    - target stk_p2_s18_t7 (Cartesian target) at (974.5, -259.38, 673.26) mm, rotated rx -64.06 ry 82.47 rz -57.48 deg; joints [17.675, -65.878, 133.528, 25.602, -72.986, -2.699] of KR 8 1620 ARC HW
    - target stk_p2_s18_t8 (Cartesian target) at (974.72, -248.82, 673.38) mm, rotated rx -62.73 ry 82.82 rz -56.53 deg; joints [16.995, -66.047, 133.813, 24.489, -72.919, -2.65] of KR 8 1620 ARC HW
    - target stk_p2_s18_t9 (Cartesian target) at (974.93, -238.26, 673.5) mm, rotated rx -61.27 ry 83.16 rz -55.44 deg; joints [16.309, -66.209, 134.087, 23.369, -72.854, -2.602] of KR 8 1620 ARC HW
    - target stk_p2_s18_t10 (Cartesian target) at (975.15, -227.7, 673.63) mm, rotated rx -59.65 ry 83.5 rz -54.2 deg; joints [15.619, -66.365, 134.348, 22.243, -72.793, -2.556] of KR 8 1620 ARC HW
    - target stk_p2_s18_t11 (Cartesian target) at (975.37, -217.15, 673.75) mm, rotated rx -57.85 ry 83.83 rz -52.78 deg; joints [14.924, -66.514, 134.596, 21.111, -72.734, -2.512] of KR 8 1620 ARC HW
    - target stk_p2_s18_t12 (Cartesian target) at (975.59, -206.59, 673.87) mm, rotated rx -55.85 ry 84.16 rz -51.15 deg; joints [14.225, -66.656, 134.833, 19.974, -72.677, -2.468] of KR 8 1620 ARC HW
    - target stk_p2_s18_t13 (Cartesian target) at (975.81, -196.03, 674) mm, rotated rx -53.61 ry 84.48 rz -49.29 deg; joints [13.522, -66.791, 135.056, 18.832, -72.624, -2.426] of KR 8 1620 ARC HW
    - target stk_p2_s18_t14 (Cartesian target) at (976.03, -185.47, 674.12) mm, rotated rx -51.1 ry 84.79 rz -47.16 deg; joints [12.814, -66.92, 135.267, 17.684, -72.573, -2.385] of KR 8 1620 ARC HW
    - target stk_p2_s18_t15 (Cartesian target) at (976.25, -174.91, 674.24) mm, rotated rx -48.28 ry 85.09 rz -44.71 deg; joints [12.103, -67.041, 135.466, 16.531, -72.525, -2.344] of KR 8 1620 ARC HW
    - target stk_p2_s18_t16 (Cartesian target) at (976.47, -164.35, 674.37) mm, rotated rx -45.1 ry 85.37 rz -41.91 deg; joints [11.388, -67.155, 135.652, 15.374, -72.479, -2.305] of KR 8 1620 ARC HW
    - target stk_p2_s18_t17 (Cartesian target) at (976.69, -153.8, 674.49) mm, rotated rx -41.5 ry 85.64 rz -38.69 deg; joints [10.669, -67.262, 135.825, 14.213, -72.437, -2.266] of KR 8 1620 ARC HW
    - target stk_p2_s18_t18 (Cartesian target) at (976.91, -143.24, 674.61) mm, rotated rx -37.45 ry 85.89 rz -35.02 deg; joints [9.947, -67.362, 135.985, 13.048, -72.397, -2.228] of KR 8 1620 ARC HW
    - target stk_p2_s18_t19 (Cartesian target) at (977.13, -132.68, 674.74) mm, rotated rx -32.89 ry 86.12 rz -30.84 deg; joints [9.223, -67.455, 136.132, 11.878, -72.359, -2.191] of KR 8 1620 ARC HW
    - target stk_p2_s18_t20 (Cartesian target) at (977.35, -122.12, 674.86) mm, rotated rx -27.79 ry 86.32 rz -26.12 deg; joints [8.495, -67.54, 136.267, 10.706, -72.324, -2.154] of KR 8 1620 ARC HW
    - target stk_p2_s18_t21 (Cartesian target) at (977.57, -111.56, 674.99) mm, rotated rx -22.15 ry 86.49 rz -20.87 deg; joints [7.765, -67.618, 136.388, 9.53, -72.292, -2.118] of KR 8 1620 ARC HW
    - target stk_p2_s18_t22 (Cartesian target) at (977.79, -101, 675.11) mm, rotated rx -16.01 ry 86.62 rz -15.1 deg; joints [7.032, -67.689, 136.497, 8.351, -72.263, -2.082] of KR 8 1620 ARC HW
    - target stk_p2_s18_t23 (Cartesian target) at (978.01, -90.44, 675.23) mm, rotated rx -9.44 ry 86.71 rz -8.92 deg; joints [6.298, -67.752, 136.592, 7.17, -72.236, -2.047] of KR 8 1620 ARC HW
    - target stk_p2_s18_t24 (Cartesian target) at (978.22, -79.89, 675.36) mm, rotated rx -2.6 ry 86.76 rz -2.46 deg; joints [5.561, -67.807, 136.675, 5.986, -72.212, -2.011] of KR 8 1620 ARC HW
    - target stk_p2_s18_t25 (Cartesian target) at (978.44, -69.33, 675.48) mm, rotated rx 4.34 ry 86.76 rz 4.1 deg; joints [4.823, -67.856, 136.745, 4.801, -72.191, -1.976] of KR 8 1620 ARC HW
    - target stk_p2_s19_t0 (Cartesian target) at (980.09, -20.25, 992.92) mm, rotated rx 166.42 ry 81.24 rz 164.19 deg; joints [1.382, -82.788, 120.669, -1.392, -29.376, -0.961] of KR 8 1620 ARC HW
    - target stk_p2_s19_t0 (Cartesian target) at (980.09, -20.25, 992.92) mm, rotated rx 166.42 ry 81.24 rz 164.19 deg; joints [1.382, -82.788, 120.669, -1.392, -29.376, -0.961] of KR 8 1620 ARC HW
    - target stk_p2_s19_t1 (Cartesian target) at (980.31, -9.7, 993.04) mm, rotated rx 163.97 ry 81.14 rz 161.32 deg; joints [0.646, -82.79, 120.662, -3.667, -29.403, 0.461] of KR 8 1620 ARC HW
    - target stk_p2_s19_t2 (Cartesian target) at (980.53, 0.86, 993.17) mm, rotated rx 161.59 ry 81.02 rz 158.52 deg; joints [-0.09, -82.781, 120.643, -5.935, -29.465, 1.877] of KR 8 1620 ARC HW
    - target stk_p2_s19_t3 (Cartesian target) at (980.75, 11.42, 993.29) mm, rotated rx 159.27 ry 80.89 rz 155.78 deg; joints [-0.826, -82.763, 120.613, -8.193, -29.56, 3.283] of KR 8 1620 ARC HW
    - target stk_p2_s19_t4 (Cartesian target) at (980.97, 21.98, 993.41) mm, rotated rx 157.02 ry 80.74 rz 153.11 deg; joints [-1.561, -82.735, 120.571, -10.434, -29.689, 4.673] of KR 8 1620 ARC HW
    - target stk_p2_s19_t5 (Cartesian target) at (981.19, 32.54, 993.54) mm, rotated rx 154.85 ry 80.58 rz 150.52 deg; joints [-2.295, -82.696, 120.518, -12.654, -29.85, 6.042] of KR 8 1620 ARC HW
    - target stk_p2_s19_t6 (Cartesian target) at (981.41, 43.1, 993.66) mm, rotated rx 152.76 ry 80.4 rz 148 deg; joints [-3.028, -82.648, 120.453, -14.85, -30.044, 7.388] of KR 8 1620 ARC HW
    - target stk_p2_s19_t7 (Cartesian target) at (981.63, 53.65, 993.78) mm, rotated rx 150.74 ry 80.21 rz 145.56 deg; joints [-3.76, -82.589, 120.376, -17.016, -30.269, 8.706] of KR 8 1620 ARC HW
    - target stk_p2_s19_t8 (Cartesian target) at (981.85, 64.21, 993.91) mm, rotated rx 148.8 ry 80.02 rz 143.2 deg; joints [-4.489, -82.521, 120.288, -19.15, -30.525, 9.992] of KR 8 1620 ARC HW
    - target stk_p2_s19_t9 (Cartesian target) at (982.07, 74.77, 994.03) mm, rotated rx 146.94 ry 79.81 rz 140.92 deg; joints [-5.218, -82.442, 120.188, -21.248, -30.81, 11.243] of KR 8 1620 ARC HW
    - target stk_p2_s19_t10 (Cartesian target) at (982.29, 85.33, 994.15) mm, rotated rx 145.16 ry 79.59 rz 138.72 deg; joints [-5.943, -82.354, 120.077, -23.307, -31.124, 12.457] of KR 8 1620 ARC HW
    - target stk_p2_s19_t11 (Cartesian target) at (982.5, 95.89, 994.28) mm, rotated rx 143.45 ry 79.36 rz 136.59 deg; joints [-6.667, -82.256, 119.954, -25.325, -31.465, 13.632] of KR 8 1620 ARC HW
    - target stk_p2_s19_t12 (Cartesian target) at (982.72, 106.45, 994.4) mm, rotated rx 141.82 ry 79.13 rz 134.54 deg; joints [-7.388, -82.148, 119.82, -27.301, -31.831, 14.766] of KR 8 1620 ARC HW
    - target stk_p2_s19_t13 (Cartesian target) at (982.94, 117.01, 994.52) mm, rotated rx 140.26 ry 78.88 rz 132.56 deg; joints [-8.106, -82.031, 119.674, -29.232, -32.222, 15.858] of KR 8 1620 ARC HW
    - target stk_p2_s19_t14 (Cartesian target) at (983.16, 127.56, 994.65) mm, rotated rx 138.76 ry 78.63 rz 130.65 deg; joints [-8.821, -81.904, 119.517, -31.118, -32.637, 16.906] of KR 8 1620 ARC HW
    - target stk_p2_s19_t15 (Cartesian target) at (983.38, 138.12, 994.77) mm, rotated rx 137.34 ry 78.38 rz 128.81 deg; joints [-9.533, -81.768, 119.348, -32.958, -33.073, 17.91] of KR 8 1620 ARC HW
    - target stk_p2_s19_t16 (Cartesian target) at (983.6, 148.68, 994.89) mm, rotated rx 135.98 ry 78.11 rz 127.03 deg; joints [-10.241, -81.622, 119.167, -34.751, -33.531, 18.869] of KR 8 1620 ARC HW
    - target stk_p2_s19_t17 (Cartesian target) at (983.82, 159.24, 995.02) mm, rotated rx 134.68 ry 77.84 rz 125.32 deg; joints [-10.946, -81.466, 118.975, -36.498, -34.008, 19.785] of KR 8 1620 ARC HW
    - target stk_p2_s19_t18 (Cartesian target) at (984.04, 169.8, 995.14) mm, rotated rx 133.43 ry 77.57 rz 123.66 deg; joints [-11.647, -81.302, 118.772, -38.198, -34.503, 20.657] of KR 8 1620 ARC HW
    - target stk_p2_s19_t19 (Cartesian target) at (984.26, 180.36, 995.27) mm, rotated rx 132.25 ry 77.29 rz 122.06 deg; joints [-12.344, -81.128, 118.557, -39.852, -35.015, 21.485] of KR 8 1620 ARC HW
    - target stk_p2_s19_t20 (Cartesian target) at (984.48, 190.91, 995.39) mm, rotated rx 131.11 ry 77 rz 120.51 deg; joints [-13.036, -80.945, 118.33, -41.461, -35.542, 22.271] of KR 8 1620 ARC HW
    - target stk_p2_s19_t21 (Cartesian target) at (984.7, 201.47, 995.51) mm, rotated rx 130.03 ry 76.71 rz 119.02 deg; joints [-13.725, -80.753, 118.092, -43.024, -36.084, 23.015] of KR 8 1620 ARC HW
    - target stk_p2_s19_t22 (Cartesian target) at (984.92, 212.03, 995.64) mm, rotated rx 128.99 ry 76.42 rz 117.57 deg; joints [-14.408, -80.553, 117.842, -44.544, -36.64, 23.718] of KR 8 1620 ARC HW
    - target stk_p2_s19_t23 (Cartesian target) at (985.14, 222.59, 995.76) mm, rotated rx 128 ry 76.12 rz 116.17 deg; joints [-15.087, -80.343, 117.581, -46.021, -37.208, 24.382] of KR 8 1620 ARC HW
    - target stk_p2_s19_t24 (Cartesian target) at (985.36, 233.15, 995.88) mm, rotated rx 127.06 ry 75.83 rz 114.81 deg; joints [-15.761, -80.125, 117.309, -47.456, -37.787, 25.008] of KR 8 1620 ARC HW
    - target stk_p2_s19_t25 (Cartesian target) at (985.58, 243.71, 996.01) mm, rotated rx 126.15 ry 75.52 rz 113.5 deg; joints [-16.43, -79.898, 117.025, -48.85, -38.376, 25.597] of KR 8 1620 ARC HW
    - target stk_p2_s20_t0 (Cartesian target) at (973.51, -337.01, 989.21) mm, rotated rx -130.97 ry 77.39 rz -120.69 deg; joints [22.363, -78.272, 115.517, 53.029, -40.963, -30.398] of KR 8 1620 ARC HW
    - target stk_p2_s20_t0 (Cartesian target) at (973.51, -337.01, 989.21) mm, rotated rx -130.97 ry 77.39 rz -120.69 deg; joints [22.363, -78.272, 115.517, 53.029, -40.963, -30.398] of KR 8 1620 ARC HW
    - target stk_p2_s20_t1 (Cartesian target) at (973.73, -326.45, 989.34) mm, rotated rx -132.16 ry 77.66 rz -122.29 deg; joints [21.726, -78.55, 115.855, 51.798, -40.347, -29.959] of KR 8 1620 ARC HW
    - target stk_p2_s20_t2 (Cartesian target) at (973.95, -315.89, 989.46) mm, rotated rx -133.41 ry 77.93 rz -123.94 deg; joints [21.084, -78.821, 116.182, 50.533, -39.738, -29.489] of KR 8 1620 ARC HW
    - target stk_p2_s20_t3 (Cartesian target) at (974.17, -305.33, 989.58) mm, rotated rx -134.71 ry 78.2 rz -125.65 deg; joints [20.436, -79.083, 116.497, 49.231, -39.135, -28.988] of KR 8 1620 ARC HW
    - target stk_p2_s20_t4 (Cartesian target) at (974.39, -294.77, 989.71) mm, rotated rx -136.07 ry 78.46 rz -127.42 deg; joints [19.783, -79.337, 116.8, 47.892, -38.541, -28.453] of KR 8 1620 ARC HW
    - target stk_p2_s20_t5 (Cartesian target) at (974.61, -284.21, 989.83) mm, rotated rx -137.5 ry 78.71 rz -129.26 deg; joints [19.124, -79.583, 117.093, 46.515, -37.955, -27.884] of KR 8 1620 ARC HW
    - target stk_p2_s20_t6 (Cartesian target) at (974.83, -273.66, 989.95) mm, rotated rx -139 ry 78.95 rz -131.17 deg; joints [18.46, -79.821, 117.374, 45.098, -37.378, -27.279] of KR 8 1620 ARC HW
    - target stk_p2_s20_t7 (Cartesian target) at (975.05, -263.1, 990.08) mm, rotated rx -140.57 ry 79.19 rz -133.15 deg; joints [17.791, -80.05, 117.643, 43.64, -36.812, -26.637] of KR 8 1620 ARC HW
    - target stk_p2_s20_t8 (Cartesian target) at (975.27, -252.54, 990.2) mm, rotated rx -142.2 ry 79.43 rz -135.2 deg; joints [17.116, -80.271, 117.901, 42.14, -36.258, -25.955] of KR 8 1620 ARC HW
    - target stk_p2_s20_t9 (Cartesian target) at (975.49, -241.98, 990.32) mm, rotated rx -143.91 ry 79.65 rz -137.32 deg; joints [16.437, -80.484, 118.148, 40.597, -35.716, -25.234] of KR 8 1620 ARC HW
    - target stk_p2_s20_t10 (Cartesian target) at (975.71, -231.42, 990.45) mm, rotated rx -145.7 ry 79.86 rz -139.53 deg; joints [15.754, -80.687, 118.383, 39.01, -35.188, -24.472] of KR 8 1620 ARC HW
    - target stk_p2_s20_t11 (Cartesian target) at (975.93, -220.86, 990.57) mm, rotated rx -147.57 ry 80.07 rz -141.81 deg; joints [15.065, -80.882, 118.606, 37.378, -34.675, -23.668] of KR 8 1620 ARC HW
    - target stk_p2_s20_t12 (Cartesian target) at (976.14, -210.31, 990.69) mm, rotated rx -149.51 ry 80.26 rz -144.16 deg; joints [14.373, -81.068, 118.819, 35.7, -34.178, -22.821] of KR 8 1620 ARC HW
    - target stk_p2_s20_t13 (Cartesian target) at (976.36, -199.75, 990.82) mm, rotated rx -151.53 ry 80.44 rz -146.6 deg; joints [13.676, -81.244, 119.019, 33.976, -33.698, -21.93] of KR 8 1620 ARC HW
    - target stk_p2_s20_t14 (Cartesian target) at (976.58, -189.19, 990.94) mm, rotated rx -153.63 ry 80.61 rz -149.12 deg; joints [12.975, -81.412, 119.209, 32.206, -33.237, -20.996] of KR 8 1620 ARC HW
    - target stk_p2_s20_t15 (Cartesian target) at (976.8, -178.63, 991.06) mm, rotated rx -155.8 ry 80.77 rz -151.71 deg; joints [12.27, -81.57, 119.386, 30.39, -32.795, -20.017] of KR 8 1620 ARC HW
    - target stk_p2_s20_t16 (Cartesian target) at (977.02, -168.07, 991.19) mm, rotated rx -158.06 ry 80.91 rz -154.38 deg; joints [11.561, -81.719, 119.553, 28.527, -32.375, -18.994] of KR 8 1620 ARC HW
    - target stk_p2_s20_t17 (Cartesian target) at (977.24, -157.51, 991.31) mm, rotated rx -160.38 ry 81.04 rz -157.12 deg; joints [10.849, -81.859, 119.707, 26.619, -31.977, -17.927] of KR 8 1620 ARC HW
    - target stk_p2_s20_t18 (Cartesian target) at (977.46, -146.96, 991.44) mm, rotated rx -162.76 ry 81.16 rz -159.93 deg; joints [10.134, -81.989, 119.851, 24.665, -31.603, -16.817] of KR 8 1620 ARC HW
    - target stk_p2_s20_t19 (Cartesian target) at (977.68, -136.4, 991.56) mm, rotated rx -165.21 ry 81.26 rz -162.8 deg; joints [9.416, -82.11, 119.982, 22.669, -31.254, -15.666] of KR 8 1620 ARC HW
    - target stk_p2_s20_t20 (Cartesian target) at (977.9, -125.84, 991.68) mm, rotated rx -167.71 ry 81.34 rz -165.72 deg; joints [8.695, -82.221, 120.103, 20.631, -30.931, -14.474] of KR 8 1620 ARC HW
    - target stk_p2_s20_t21 (Cartesian target) at (978.12, -115.28, 991.81) mm, rotated rx -170.26 ry 81.41 rz -168.69 deg; joints [7.971, -82.322, 120.211, 18.553, -30.635, -13.243] of KR 8 1620 ARC HW
    - target stk_p2_s20_t22 (Cartesian target) at (978.34, -104.72, 991.93) mm, rotated rx -172.85 ry 81.46 rz -171.7 deg; joints [7.245, -82.413, 120.308, 16.437, -30.369, -11.977] of KR 8 1620 ARC HW
    - target stk_p2_s20_t23 (Cartesian target) at (978.56, -94.16, 992.05) mm, rotated rx -175.46 ry 81.5 rz -174.73 deg; joints [6.517, -82.495, 120.394, 14.288, -30.132, -10.677] of KR 8 1620 ARC HW
    - target stk_p2_s20_t24 (Cartesian target) at (978.78, -83.6, 992.18) mm, rotated rx -178.09 ry 81.51 rz -177.78 deg; joints [5.787, -82.567, 120.468, 12.107, -29.925, -9.347] of KR 8 1620 ARC HW
    - target stk_p2_s20_t25 (Cartesian target) at (979, -73.05, 992.3) mm, rotated rx 179.28 ry 81.51 rz 179.17 deg; joints [5.056, -82.629, 120.53, 9.9, -29.751, -7.991] of KR 8 1620 ARC HW
    - target stk_p3_s21_t0 (Cartesian target) at (979.69, -17.53, 760.58) mm, rotated rx 88.12 ry 87.83 rz 85.95 deg; joints [0.159, -73.03, 133.853, -2.305, -60.913, -1.05] of KR 8 1620 ARC HW
    - target stk_p3_s21_t0 (Cartesian target) at (979.69, -17.53, 760.58) mm, rotated rx 88.12 ry 87.83 rz 85.95 deg; joints [0.159, -73.03, 133.853, -2.305, -60.913, -1.05] of KR 8 1620 ARC HW
    - target stk_p3_s21_t1 (Cartesian target) at (979.91, -6.97, 760.71) mm, rotated rx 88.51 ry 87.43 rz 85.95 deg; joints [-0.582, -73.021, 133.814, -3.603, -60.908, -0.808] of KR 8 1620 ARC HW
    - target stk_p3_s21_t2 (Cartesian target) at (980.13, 3.59, 760.83) mm, rotated rx 88.8 ry 87.04 rz 85.84 deg; joints [-1.323, -73.002, 133.762, -4.901, -60.911, -0.567] of KR 8 1620 ARC HW
    - target stk_p3_s21_t3 (Cartesian target) at (980.35, 14.15, 760.95) mm, rotated rx 89.02 ry 86.65 rz 85.67 deg; joints [-2.063, -72.975, 133.697, -6.197, -60.922, -0.324] of KR 8 1620 ARC HW
    - target stk_p3_s21_t4 (Cartesian target) at (980.56, 24.71, 761.08) mm, rotated rx 89.19 ry 86.26 rz 85.45 deg; joints [-2.801, -72.94, 133.619, -7.492, -60.942, -0.082] of KR 8 1620 ARC HW
    - target stk_p3_s21_t5 (Cartesian target) at (980.78, 35.26, 761.2) mm, rotated rx 89.33 ry 85.86 rz 85.2 deg; joints [-3.538, -72.895, 133.529, -8.784, -60.97, 0.16] of KR 8 1620 ARC HW
    - target stk_p3_s21_t6 (Cartesian target) at (981, 45.82, 761.32) mm, rotated rx 89.45 ry 85.47 rz 84.92 deg; joints [-4.273, -72.843, 133.426, -10.073, -61.007, 0.401] of KR 8 1620 ARC HW
    - target stk_p3_s21_t7 (Cartesian target) at (981.22, 56.38, 761.45) mm, rotated rx 89.55 ry 85.08 rz 84.63 deg; joints [-5.006, -72.781, 133.311, -11.359, -61.051, 0.642] of KR 8 1620 ARC HW
    - target stk_p3_s21_t8 (Cartesian target) at (981.44, 66.94, 761.57) mm, rotated rx 89.63 ry 84.69 rz 84.32 deg; joints [-5.736, -72.712, 133.182, -12.64, -61.104, 0.882] of KR 8 1620 ARC HW
    - target stk_p3_s21_t9 (Cartesian target) at (981.66, 77.5, 761.69) mm, rotated rx 89.7 ry 84.3 rz 84 deg; joints [-6.464, -72.634, 133.042, -13.918, -61.165, 1.122] of KR 8 1620 ARC HW
    - target stk_p3_s21_t10 (Cartesian target) at (981.88, 88.06, 761.82) mm, rotated rx 89.76 ry 83.91 rz 83.67 deg; joints [-7.189, -72.547, 132.888, -15.19, -61.235, 1.36] of KR 8 1620 ARC HW
    - target stk_p3_s21_t11 (Cartesian target) at (982.1, 98.62, 761.94) mm, rotated rx 89.82 ry 83.52 rz 83.34 deg; joints [-7.911, -72.452, 132.722, -16.458, -61.312, 1.597] of KR 8 1620 ARC HW
    - target stk_p3_s21_t12 (Cartesian target) at (982.32, 109.17, 762.07) mm, rotated rx 89.87 ry 83.13 rz 83 deg; joints [-8.629, -72.35, 132.544, -17.72, -61.397, 1.832] of KR 8 1620 ARC HW
    - target stk_p3_s21_t13 (Cartesian target) at (982.54, 119.73, 762.19) mm, rotated rx 89.91 ry 82.74 rz 82.65 deg; joints [-9.344, -72.238, 132.353, -18.975, -61.49, 2.066] of KR 8 1620 ARC HW
    - target stk_p3_s21_t14 (Cartesian target) at (982.76, 130.29, 762.31) mm, rotated rx 89.95 ry 82.35 rz 82.3 deg; joints [-10.055, -72.119, 132.15, -20.224, -61.59, 2.298] of KR 8 1620 ARC HW
    - target stk_p3_s21_t15 (Cartesian target) at (982.98, 140.85, 762.44) mm, rotated rx 89.98 ry 81.97 rz 81.95 deg; joints [-10.763, -71.992, 131.935, -21.467, -61.698, 2.528] of KR 8 1620 ARC HW
    - target stk_p3_s21_t16 (Cartesian target) at (983.2, 151.41, 762.56) mm, rotated rx 90.02 ry 81.58 rz 81.59 deg; joints [-11.466, -71.857, 131.707, -22.702, -61.813, 2.756] of KR 8 1620 ARC HW
    - target stk_p3_s21_t17 (Cartesian target) at (983.42, 161.97, 762.68) mm, rotated rx 90.05 ry 81.19 rz 81.24 deg; joints [-12.165, -71.714, 131.467, -23.929, -61.936, 2.982] of KR 8 1620 ARC HW
    - target stk_p3_s21_t18 (Cartesian target) at (983.64, 172.52, 762.81) mm, rotated rx 90.07 ry 80.81 rz 80.88 deg; joints [-12.86, -71.563, 131.215, -25.149, -62.066, 3.206] of KR 8 1620 ARC HW
    - target stk_p3_s21_t19 (Cartesian target) at (983.85, 183.08, 762.93) mm, rotated rx 90.1 ry 80.42 rz 80.52 deg; joints [-13.55, -71.405, 130.951, -26.361, -62.203, 3.428] of KR 8 1620 ARC HW
    - target stk_p3_s21_t20 (Cartesian target) at (984.07, 193.64, 763.05) mm, rotated rx 90.12 ry 80.04 rz 80.15 deg; joints [-14.235, -71.239, 130.675, -27.563, -62.346, 3.647] of KR 8 1620 ARC HW
    - target stk_p3_s21_t21 (Cartesian target) at (984.29, 204.2, 763.18) mm, rotated rx 90.14 ry 79.65 rz 79.79 deg; joints [-14.915, -71.065, 130.387, -28.758, -62.496, 3.864] of KR 8 1620 ARC HW
    - target stk_p3_s21_t22 (Cartesian target) at (984.51, 214.76, 763.3) mm, rotated rx 90.16 ry 79.27 rz 79.43 deg; joints [-15.59, -70.884, 130.087, -29.943, -62.653, 4.079] of KR 8 1620 ARC HW
    - target stk_p3_s21_t23 (Cartesian target) at (984.73, 225.32, 763.42) mm, rotated rx 90.18 ry 78.89 rz 79.06 deg; joints [-16.259, -70.696, 129.775, -31.118, -62.816, 4.291] of KR 8 1620 ARC HW
    - target stk_p3_s21_t24 (Cartesian target) at (984.95, 235.88, 763.55) mm, rotated rx 90.19 ry 78.51 rz 78.7 deg; joints [-16.924, -70.5, 129.451, -32.284, -62.986, 4.5] of KR 8 1620 ARC HW
    - target stk_p3_s21_t25 (Cartesian target) at (985.17, 246.43, 763.67) mm, rotated rx 90.21 ry 78.13 rz 78.33 deg; joints [-17.583, -70.298, 129.116, -33.441, -63.161, 4.708] of KR 8 1620 ARC HW
    - target stk_p3_s22_t0 (Cartesian target) at (973.11, -334.28, 756.88) mm, rotated rx -88.75 ry 80.51 rz -79.28 deg; joints [21.555, -69.45, 129.11, 34.827, -64.553, -7.278] of KR 8 1620 ARC HW
    - target stk_p3_s22_t0 (Cartesian target) at (973.11, -334.28, 756.88) mm, rotated rx -88.75 ry 80.51 rz -79.28 deg; joints [21.555, -69.45, 129.11, 34.827, -64.553, -7.278] of KR 8 1620 ARC HW
    - target stk_p3_s22_t1 (Cartesian target) at (973.33, -323.72, 757) mm, rotated rx -88.73 ry 80.89 rz -79.64 deg; joints [20.901, -69.681, 129.449, 33.7, -64.344, -7.114] of KR 8 1620 ARC HW
    - target stk_p3_s22_t2 (Cartesian target) at (973.55, -313.16, 757.12) mm, rotated rx -88.7 ry 81.27 rz -79.99 deg; joints [20.24, -69.905, 129.775, 32.562, -64.139, -6.946] of KR 8 1620 ARC HW
    - target stk_p3_s22_t3 (Cartesian target) at (973.77, -302.6, 757.25) mm, rotated rx -88.67 ry 81.65 rz -80.34 deg; joints [19.574, -70.122, 130.09, 31.415, -63.939, -6.776] of KR 8 1620 ARC HW
    - target stk_p3_s22_t4 (Cartesian target) at (973.99, -292.05, 757.37) mm, rotated rx -88.64 ry 82.03 rz -80.69 deg; joints [18.903, -70.332, 130.392, 30.258, -63.745, -6.602] of KR 8 1620 ARC HW
    - target stk_p3_s22_t5 (Cartesian target) at (974.2, -281.49, 757.49) mm, rotated rx -88.61 ry 82.42 rz -81.04 deg; joints [18.226, -70.535, 130.682, 29.092, -63.555, -6.426] of KR 8 1620 ARC HW
    - target stk_p3_s22_t6 (Cartesian target) at (974.42, -270.93, 757.62) mm, rotated rx -88.57 ry 82.8 rz -81.38 deg; joints [17.544, -70.73, 130.96, 27.916, -63.37, -6.246] of KR 8 1620 ARC HW
    - target stk_p3_s22_t7 (Cartesian target) at (974.64, -260.37, 757.74) mm, rotated rx -88.52 ry 83.19 rz -81.72 deg; joints [16.858, -70.918, 131.225, 26.731, -63.19, -6.063] of KR 8 1620 ARC HW
    - target stk_p3_s22_t8 (Cartesian target) at (974.86, -249.81, 757.86) mm, rotated rx -88.47 ry 83.57 rz -82.06 deg; joints [16.166, -71.099, 131.478, 25.537, -63.016, -5.877] of KR 8 1620 ARC HW
    - target stk_p3_s22_t9 (Cartesian target) at (975.08, -239.25, 757.99) mm, rotated rx -88.42 ry 83.96 rz -82.39 deg; joints [15.47, -71.272, 131.719, 24.334, -62.848, -5.687] of KR 8 1620 ARC HW
    - target stk_p3_s22_t10 (Cartesian target) at (975.3, -228.7, 758.11) mm, rotated rx -88.36 ry 84.35 rz -82.71 deg; joints [14.77, -71.437, 131.947, 23.124, -62.686, -5.495] of KR 8 1620 ARC HW
    - target stk_p3_s22_t11 (Cartesian target) at (975.52, -218.14, 758.24) mm, rotated rx -88.28 ry 84.73 rz -83.03 deg; joints [14.065, -71.595, 132.163, 21.905, -62.529, -5.299] of KR 8 1620 ARC HW
    - target stk_p3_s22_t12 (Cartesian target) at (975.74, -207.58, 758.36) mm, rotated rx -88.2 ry 85.12 rz -83.33 deg; joints [13.356, -71.745, 132.367, 20.678, -62.379, -5.099] of KR 8 1620 ARC HW
    - target stk_p3_s22_t13 (Cartesian target) at (975.96, -197.02, 758.48) mm, rotated rx -88.1 ry 85.51 rz -83.62 deg; joints [12.643, -71.887, 132.558, 19.444, -62.235, -4.897] of KR 8 1620 ARC HW
    - target stk_p3_s22_t14 (Cartesian target) at (976.18, -186.46, 758.61) mm, rotated rx -87.98 ry 85.9 rz -83.89 deg; joints [11.927, -72.021, 132.736, 18.202, -62.098, -4.691] of KR 8 1620 ARC HW
    - target stk_p3_s22_t15 (Cartesian target) at (976.4, -175.9, 758.73) mm, rotated rx -87.84 ry 86.29 rz -84.14 deg; joints [11.207, -72.147, 132.901, 16.954, -61.968, -4.482] of KR 8 1620 ARC HW
    - target stk_p3_s22_t16 (Cartesian target) at (976.62, -165.35, 758.85) mm, rotated rx -87.67 ry 86.68 rz -84.35 deg; joints [10.484, -72.265, 133.054, 15.7, -61.844, -4.27] of KR 8 1620 ARC HW
    - target stk_p3_s22_t17 (Cartesian target) at (976.84, -154.79, 758.98) mm, rotated rx -87.44 ry 87.07 rz -84.52 deg; joints [9.758, -72.375, 133.194, 14.439, -61.728, -4.055] of KR 8 1620 ARC HW
    - target stk_p3_s22_t18 (Cartesian target) at (977.06, -144.23, 759.1) mm, rotated rx -87.15 ry 87.46 rz -84.62 deg; joints [9.029, -72.476, 133.322, 13.173, -61.618, -3.837] of KR 8 1620 ARC HW
    - target stk_p3_s22_t19 (Cartesian target) at (977.28, -133.67, 759.22) mm, rotated rx -86.76 ry 87.85 rz -84.61 deg; joints [8.298, -72.569, 133.437, 11.901, -61.516, -3.617] of KR 8 1620 ARC HW
    - target stk_p3_s22_t20 (Cartesian target) at (977.49, -123.11, 759.35) mm, rotated rx -86.18 ry 88.24 rz -84.43 deg; joints [7.565, -72.654, 133.539, 10.625, -61.422, -3.394] of KR 8 1620 ARC HW
    - target stk_p3_s22_t21 (Cartesian target) at (977.71, -112.55, 759.47) mm, rotated rx -85.28 ry 88.63 rz -83.92 deg; joints [6.829, -72.73, 133.628, 9.344, -61.335, -3.168] of KR 8 1620 ARC HW
    - target stk_p3_s22_t22 (Cartesian target) at (977.93, -101.99, 759.59) mm, rotated rx -83.65 ry 89.02 rz -82.68 deg; joints [6.091, -72.798, 133.704, 8.059, -61.256, -2.94] of KR 8 1620 ARC HW
    - target stk_p3_s22_t23 (Cartesian target) at (978.15, -91.44, 759.72) mm, rotated rx -79.84 ry 89.41 rz -79.27 deg; joints [5.353, -72.857, 133.768, 6.771, -61.184, -2.709] of KR 8 1620 ARC HW
    - target stk_p3_s22_t24 (Cartesian target) at (978.37, -80.88, 759.84) mm, rotated rx -61.79 ry 89.79 rz -61.6 deg; joints [4.612, -72.908, 133.818, 5.48, -61.121, -2.477] of KR 8 1620 ARC HW
    - target stk_p3_s22_t25 (Cartesian target) at (978.59, -70.32, 759.97) mm, rotated rx 65.72 ry 89.77 rz 65.51 deg; joints [3.871, -72.95, 133.856, 4.186, -61.066, -2.243] of KR 8 1620 ARC HW
    - target stk_p3_s23_t0 (Cartesian target) at (979.87, -18.77, 866.19) mm, rotated rx 151.13 ry 85.6 rz 148.93 deg; joints [0.249, -78.342, 128.735, -2.582, -46.569, -0.478] of KR 8 1620 ARC HW
    - target stk_p3_s23_t0 (Cartesian target) at (979.87, -18.77, 866.19) mm, rotated rx 151.13 ry 85.6 rz 148.93 deg; joints [0.249, -78.342, 128.735, -2.582, -46.569, -0.478] of KR 8 1620 ARC HW
    - target stk_p3_s23_t1 (Cartesian target) at (980.09, -8.21, 866.31) mm, rotated rx 146.88 ry 85.39 rz 144.28 deg; joints [-0.492, -78.328, 128.696, -4.139, -46.582, 0.124] of KR 8 1620 ARC HW
    - target stk_p3_s23_t2 (Cartesian target) at (980.31, 2.35, 866.44) mm, rotated rx 143.02 ry 85.17 rz 140 deg; joints [-1.231, -78.304, 128.645, -5.693, -46.612, 0.726] of KR 8 1620 ARC HW
    - target stk_p3_s23_t3 (Cartesian target) at (980.53, 12.91, 866.56) mm, rotated rx 139.51 ry 84.92 rz 136.1 deg; joints [-1.969, -78.271, 128.581, -7.245, -46.659, 1.325] of KR 8 1620 ARC HW
    - target stk_p3_s23_t4 (Cartesian target) at (980.75, 23.47, 866.68) mm, rotated rx 136.35 ry 84.65 rz 132.53 deg; joints [-2.706, -78.229, 128.505, -8.792, -46.723, 1.921] of KR 8 1620 ARC HW
    - target stk_p3_s23_t5 (Cartesian target) at (980.97, 34.03, 866.81) mm, rotated rx 133.49 ry 84.37 rz 129.26 deg; joints [-3.442, -78.177, 128.417, -10.333, -46.804, 2.513] of KR 8 1620 ARC HW
    - target stk_p3_s23_t6 (Cartesian target) at (981.19, 44.58, 866.93) mm, rotated rx 130.91 ry 84.08 rz 126.28 deg; joints [-4.175, -78.115, 128.316, -11.868, -46.901, 3.1] of KR 8 1620 ARC HW
    - target stk_p3_s23_t7 (Cartesian target) at (981.41, 55.14, 867.05) mm, rotated rx 128.58 ry 83.78 rz 123.54 deg; joints [-4.906, -78.044, 128.204, -13.395, -47.014, 3.682] of KR 8 1620 ARC HW
    - target stk_p3_s23_t8 (Cartesian target) at (981.63, 65.7, 867.18) mm, rotated rx 126.47 ry 83.46 rz 121.03 deg; joints [-5.636, -77.964, 128.079, -14.913, -47.144, 4.257] of KR 8 1620 ARC HW
    - target stk_p3_s23_t9 (Cartesian target) at (981.85, 76.26, 867.3) mm, rotated rx 124.55 ry 83.14 rz 118.71 deg; joints [-6.362, -77.875, 127.942, -16.421, -47.289, 4.824] of KR 8 1620 ARC HW
    - target stk_p3_s23_t10 (Cartesian target) at (982.06, 86.82, 867.43) mm, rotated rx 122.81 ry 82.82 rz 116.56 deg; joints [-7.086, -77.777, 127.793, -17.919, -47.45, 5.384] of KR 8 1620 ARC HW
    - target stk_p3_s23_t11 (Cartesian target) at (982.28, 97.38, 867.55) mm, rotated rx 121.22 ry 82.49 rz 114.57 deg; joints [-7.806, -77.669, 127.632, -19.405, -47.626, 5.934] of KR 8 1620 ARC HW
    - target stk_p3_s23_t12 (Cartesian target) at (982.5, 107.93, 867.67) mm, rotated rx 119.77 ry 82.15 rz 112.71 deg; joints [-8.524, -77.552, 127.46, -20.878, -47.816, 6.475] of KR 8 1620 ARC HW
    - target stk_p3_s23_t13 (Cartesian target) at (982.72, 118.49, 867.8) mm, rotated rx 118.44 ry 81.81 rz 110.98 deg; joints [-9.238, -77.427, 127.275, -22.339, -48.021, 7.007] of KR 8 1620 ARC HW
    - target stk_p3_s23_t14 (Cartesian target) at (982.94, 129.05, 867.92) mm, rotated rx 117.22 ry 81.46 rz 109.36 deg; joints [-9.948, -77.292, 127.078, -23.785, -48.24, 7.527] of KR 8 1620 ARC HW
    - target stk_p3_s23_t15 (Cartesian target) at (983.16, 139.61, 868.04) mm, rotated rx 116.09 ry 81.12 rz 107.83 deg; joints [-10.654, -77.149, 126.869, -25.217, -48.472, 8.037] of KR 8 1620 ARC HW
    - target stk_p3_s23_t16 (Cartesian target) at (983.38, 150.17, 868.17) mm, rotated rx 115.05 ry 80.77 rz 106.39 deg; joints [-11.357, -76.997, 126.648, -26.634, -48.717, 8.535] of KR 8 1620 ARC HW
    - target stk_p3_s23_t17 (Cartesian target) at (983.6, 160.73, 868.29) mm, rotated rx 114.09 ry 80.42 rz 105.02 deg; joints [-12.055, -76.836, 126.416, -28.035, -48.975, 9.022] of KR 8 1620 ARC HW
    - target stk_p3_s23_t18 (Cartesian target) at (983.82, 171.28, 868.41) mm, rotated rx 113.19 ry 80.06 rz 103.73 deg; joints [-12.748, -76.667, 126.172, -29.419, -49.245, 9.497] of KR 8 1620 ARC HW
    - target stk_p3_s23_t19 (Cartesian target) at (984.04, 181.84, 868.54) mm, rotated rx 112.36 ry 79.71 rz 102.5 deg; joints [-13.437, -76.49, 125.916, -30.788, -49.526, 9.96] of KR 8 1620 ARC HW
    - target stk_p3_s23_t20 (Cartesian target) at (984.26, 192.4, 868.66) mm, rotated rx 111.59 ry 79.35 rz 101.33 deg; joints [-14.122, -76.304, 125.648, -32.139, -49.818, 10.41] of KR 8 1620 ARC HW
    - target stk_p3_s23_t21 (Cartesian target) at (984.48, 202.96, 868.78) mm, rotated rx 110.86 ry 78.99 rz 100.21 deg; joints [-14.801, -76.11, 125.368, -33.473, -50.122, 10.848] of KR 8 1620 ARC HW
    - target stk_p3_s23_t22 (Cartesian target) at (984.7, 213.52, 868.91) mm, rotated rx 110.19 ry 78.63 rz 99.14 deg; joints [-15.475, -75.908, 125.077, -34.79, -50.435, 11.273] of KR 8 1620 ARC HW
    - target stk_p3_s23_t23 (Cartesian target) at (984.92, 224.08, 869.03) mm, rotated rx 109.55 ry 78.27 rz 98.11 deg; joints [-16.144, -75.698, 124.775, -36.089, -50.758, 11.686] of KR 8 1620 ARC HW
    - target stk_p3_s23_t24 (Cartesian target) at (985.13, 234.64, 869.15) mm, rotated rx 108.95 ry 77.92 rz 97.12 deg; joints [-16.808, -75.48, 124.46, -37.371, -51.091, 12.086] of KR 8 1620 ARC HW
    - target stk_p3_s23_t25 (Cartesian target) at (985.35, 245.19, 869.28) mm, rotated rx 108.39 ry 77.56 rz 96.16 deg; joints [-17.466, -75.255, 124.135, -38.634, -51.432, 12.474] of KR 8 1620 ARC HW
    - target stk_p3_s24_t0 (Cartesian target) at (973.29, -335.52, 862.48) mm, rotated rx -111.07 ry 79.8 rz -101.23 deg; joints [21.6, -74.474, 124.219, 40.192, -53.089, -15.165] of KR 8 1620 ARC HW
    - target stk_p3_s24_t0 (Cartesian target) at (973.29, -335.52, 862.48) mm, rotated rx -111.07 ry 79.8 rz -101.23 deg; joints [21.6, -74.474, 124.219, 40.192, -53.089, -15.165] of KR 8 1620 ARC HW
    - target stk_p3_s24_t1 (Cartesian target) at (973.51, -324.96, 862.61) mm, rotated rx -111.9 ry 80.15 rz -102.45 deg; joints [20.946, -74.726, 124.545, 38.983, -52.712, -14.844] of KR 8 1620 ARC HW
    - target stk_p3_s24_t2 (Cartesian target) at (973.73, -314.4, 862.73) mm, rotated rx -112.8 ry 80.5 rz -103.74 deg; joints [20.287, -74.971, 124.859, 37.757, -52.342, -14.511] of KR 8 1620 ARC HW
    - target stk_p3_s24_t3 (Cartesian target) at (973.95, -303.84, 862.85) mm, rotated rx -113.77 ry 80.84 rz -105.1 deg; joints [19.623, -75.207, 125.161, 36.513, -51.979, -14.166] of KR 8 1620 ARC HW
    - target stk_p3_s24_t4 (Cartesian target) at (974.17, -293.29, 862.98) mm, rotated rx -114.81 ry 81.19 rz -106.54 deg; joints [18.952, -75.437, 125.451, 35.251, -51.624, -13.807] of KR 8 1620 ARC HW
    - target stk_p3_s24_t5 (Cartesian target) at (974.39, -282.73, 863.1) mm, rotated rx -115.94 ry 81.53 rz -108.07 deg; joints [18.277, -75.658, 125.729, 33.972, -51.277, -13.436] of KR 8 1620 ARC HW
    - target stk_p3_s24_t6 (Cartesian target) at (974.61, -272.17, 863.22) mm, rotated rx -117.17 ry 81.87 rz -109.69 deg; joints [17.597, -75.871, 125.996, 32.675, -50.939, -13.052] of KR 8 1620 ARC HW
    - target stk_p3_s24_t7 (Cartesian target) at (974.83, -261.61, 863.35) mm, rotated rx -118.51 ry 82.21 rz -111.43 deg; joints [16.912, -76.076, 126.25, 31.361, -50.609, -12.655] of KR 8 1620 ARC HW
    - target stk_p3_s24_t8 (Cartesian target) at (975.05, -251.05, 863.47) mm, rotated rx -119.97 ry 82.54 rz -113.29 deg; joints [16.222, -76.273, 126.492, 30.03, -50.289, -12.245] of KR 8 1620 ARC HW
    - target stk_p3_s24_t9 (Cartesian target) at (975.27, -240.49, 863.6) mm, rotated rx -121.56 ry 82.87 rz -115.28 deg; joints [15.527, -76.461, 126.722, 28.682, -49.979, -11.822] of KR 8 1620 ARC HW
    - target stk_p3_s24_t10 (Cartesian target) at (975.49, -229.94, 863.72) mm, rotated rx -123.32 ry 83.19 rz -117.43 deg; joints [14.828, -76.641, 126.941, 27.317, -49.68, -11.385] of KR 8 1620 ARC HW
    - target stk_p3_s24_t11 (Cartesian target) at (975.7, -219.38, 863.84) mm, rotated rx -125.24 ry 83.51 rz -119.76 deg; joints [14.125, -76.813, 127.147, 25.936, -49.391, -10.936] of KR 8 1620 ARC HW
    - target stk_p3_s24_t12 (Cartesian target) at (975.92, -208.82, 863.97) mm, rotated rx -127.36 ry 83.82 rz -122.28 deg; joints [13.417, -76.976, 127.34, 24.539, -49.114, -10.474] of KR 8 1620 ARC HW
    - target stk_p3_s24_t13 (Cartesian target) at (976.14, -198.26, 864.09) mm, rotated rx -129.71 ry 84.11 rz -125.03 deg; joints [12.706, -77.13, 127.522, 23.126, -48.849, -9.999] of KR 8 1620 ARC HW
    - target stk_p3_s24_t14 (Cartesian target) at (976.36, -187.7, 864.21) mm, rotated rx -132.3 ry 84.4 rz -128.02 deg; joints [11.991, -77.275, 127.692, 21.699, -48.596, -9.512] of KR 8 1620 ARC HW
    - target stk_p3_s24_t15 (Cartesian target) at (976.58, -177.14, 864.34) mm, rotated rx -135.18 ry 84.68 rz -131.3 deg; joints [11.273, -77.411, 127.849, 20.256, -48.357, -9.012] of KR 8 1620 ARC HW
    - target stk_p3_s24_t16 (Cartesian target) at (976.8, -166.58, 864.46) mm, rotated rx -138.36 ry 84.94 rz -134.88 deg; joints [10.552, -77.539, 127.994, 18.8, -48.13, -8.502] of KR 8 1620 ARC HW
    - target stk_p3_s24_t17 (Cartesian target) at (977.02, -156.03, 864.58) mm, rotated rx -141.88 ry 85.19 rz -138.81 deg; joints [9.827, -77.657, 128.127, 17.33, -47.918, -7.98] of KR 8 1620 ARC HW
    - target stk_p3_s24_t18 (Cartesian target) at (977.24, -145.47, 864.71) mm, rotated rx -145.77 ry 85.42 rz -143.1 deg; joints [9.1, -77.766, 128.247, 15.848, -47.719, -7.447] of KR 8 1620 ARC HW
    - target stk_p3_s24_t19 (Cartesian target) at (977.46, -134.91, 864.83) mm, rotated rx -150.04 ry 85.62 rz -147.78 deg; joints [8.37, -77.866, 128.356, 14.355, -47.535, -6.904] of KR 8 1620 ARC HW
    - target stk_p3_s24_t20 (Cartesian target) at (977.68, -124.35, 864.95) mm, rotated rx -154.71 ry 85.79 rz -152.85 deg; joints [7.638, -77.956, 128.452, 12.85, -47.367, -6.352] of KR 8 1620 ARC HW
    - target stk_p3_s24_t21 (Cartesian target) at (977.9, -113.79, 865.08) mm, rotated rx -159.74 ry 85.94 rz -158.29 deg; joints [6.904, -78.037, 128.536, 11.335, -47.213, -5.79] of KR 8 1620 ARC HW
    - target stk_p3_s24_t22 (Cartesian target) at (978.12, -103.23, 865.2) mm, rotated rx -165.11 ry 86.05 rz -164.06 deg; joints [6.168, -78.109, 128.607, 9.811, -47.076, -5.221] of KR 8 1620 ARC HW
    - target stk_p3_s24_t23 (Cartesian target) at (978.34, -92.68, 865.33) mm, rotated rx -170.75 ry 86.13 rz -170.11 deg; joints [5.431, -78.172, 128.666, 8.279, -46.954, -4.645] of KR 8 1620 ARC HW
    - target stk_p3_s24_t24 (Cartesian target) at (978.56, -82.12, 865.45) mm, rotated rx -176.56 ry 86.17 rz -176.32 deg; joints [4.692, -78.225, 128.713, 6.74, -46.849, -4.062] of KR 8 1620 ARC HW
    - target stk_p3_s24_t25 (Cartesian target) at (978.77, -71.56, 865.57) mm, rotated rx 177.57 ry 86.17 rz 177.4 deg; joints [3.953, -78.268, 128.747, 5.195, -46.76, -3.473] of KR 8 1620 ARC HW
    - target stk_p3_s25_t0 (Cartesian target) at (972.92, -333.04, 651.27) mm, rotated rx -66.61 ry 79.73 rz -57.5 deg; joints [21.494, -63.131, 132.613, 31.83, -76.492, -1.237] of KR 8 1620 ARC HW
    - target stk_p3_s25_t0 (Cartesian target) at (972.92, -333.04, 651.27) mm, rotated rx -66.61 ry 79.73 rz -57.5 deg; joints [21.494, -63.131, 132.613, 31.83, -76.492, -1.237] of KR 8 1620 ARC HW
    - target stk_p3_s25_t1 (Cartesian target) at (973.14, -322.48, 651.39) mm, rotated rx -65.74 ry 80.08 rz -57 deg; joints [20.839, -63.331, 132.963, 30.766, -76.433, -1.219] of KR 8 1620 ARC HW
    - target stk_p3_s25_t2 (Cartesian target) at (973.36, -311.92, 651.52) mm, rotated rx -64.81 ry 80.42 rz -56.44 deg; joints [20.177, -63.525, 133.3, 29.696, -76.375, -1.204] of KR 8 1620 ARC HW
    - target stk_p3_s25_t3 (Cartesian target) at (973.58, -301.37, 651.64) mm, rotated rx -63.81 ry 80.77 rz -55.81 deg; joints [19.51, -63.713, 133.626, 28.618, -76.319, -1.192] of KR 8 1620 ARC HW
    - target stk_p3_s25_t4 (Cartesian target) at (973.8, -290.81, 651.76) mm, rotated rx -62.74 ry 81.11 rz -55.1 deg; joints [18.838, -63.894, 133.939, 27.534, -76.265, -1.183] of KR 8 1620 ARC HW
    - target stk_p3_s25_t5 (Cartesian target) at (974.02, -280.25, 651.89) mm, rotated rx -61.57 ry 81.45 rz -54.3 deg; joints [18.161, -64.07, 134.239, 26.444, -76.213, -1.177] of KR 8 1620 ARC HW
    - target stk_p3_s25_t6 (Cartesian target) at (974.24, -269.69, 652.01) mm, rotated rx -60.31 ry 81.78 rz -53.41 deg; joints [17.478, -64.239, 134.528, 25.348, -76.162, -1.173] of KR 8 1620 ARC HW
    - target stk_p3_s25_t7 (Cartesian target) at (974.46, -259.13, 652.13) mm, rotated rx -58.94 ry 82.12 rz -52.41 deg; joints [16.79, -64.402, 134.803, 24.245, -76.112, -1.172] of KR 8 1620 ARC HW
    - target stk_p3_s25_t8 (Cartesian target) at (974.68, -248.57, 652.26) mm, rotated rx -57.44 ry 82.44 rz -51.29 deg; joints [16.098, -64.558, 135.066, 23.137, -76.064, -1.173] of KR 8 1620 ARC HW
    - target stk_p3_s25_t9 (Cartesian target) at (974.9, -238.01, 652.38) mm, rotated rx -55.81 ry 82.77 rz -50.03 deg; joints [15.401, -64.708, 135.317, 22.023, -76.017, -1.177] of KR 8 1620 ARC HW
    - target stk_p3_s25_t10 (Cartesian target) at (975.12, -227.46, 652.51) mm, rotated rx -54.02 ry 83.08 rz -48.62 deg; joints [14.7, -64.852, 135.554, 20.904, -75.972, -1.183] of KR 8 1620 ARC HW
    - target stk_p3_s25_t11 (Cartesian target) at (975.34, -216.9, 652.63) mm, rotated rx -52.07 ry 83.39 rz -47.03 deg; joints [13.994, -64.988, 135.779, 19.779, -75.928, -1.19] of KR 8 1620 ARC HW
    - target stk_p3_s25_t12 (Cartesian target) at (975.56, -206.34, 652.75) mm, rotated rx -49.92 ry 83.7 rz -45.26 deg; joints [13.284, -65.119, 135.991, 18.65, -75.885, -1.2] of KR 8 1620 ARC HW
    - target stk_p3_s25_t13 (Cartesian target) at (975.78, -195.78, 652.88) mm, rotated rx -47.55 ry 83.99 rz -43.27 deg; joints [12.57, -65.242, 136.191, 17.516, -75.844, -1.211] of KR 8 1620 ARC HW
    - target stk_p3_s25_t14 (Cartesian target) at (975.99, -185.22, 653) mm, rotated rx -44.95 ry 84.27 rz -41.04 deg; joints [11.853, -65.358, 136.377, 16.378, -75.803, -1.224] of KR 8 1620 ARC HW
    - target stk_p3_s25_t15 (Cartesian target) at (976.21, -174.66, 653.12) mm, rotated rx -42.07 ry 84.54 rz -38.54 deg; joints [11.132, -65.468, 136.55, 15.236, -75.764, -1.238] of KR 8 1620 ARC HW
    - target stk_p3_s25_t16 (Cartesian target) at (976.43, -164.11, 653.25) mm, rotated rx -38.91 ry 84.8 rz -35.75 deg; joints [10.408, -65.571, 136.71, 14.089, -75.726, -1.253] of KR 8 1620 ARC HW
    - target stk_p3_s25_t17 (Cartesian target) at (976.65, -153.55, 653.37) mm, rotated rx -35.42 ry 85.04 rz -32.64 deg; joints [9.681, -65.667, 136.857, 12.939, -75.689, -1.269] of KR 8 1620 ARC HW
    - target stk_p3_s25_t18 (Cartesian target) at (976.87, -142.99, 653.49) mm, rotated rx -31.6 ry 85.26 rz -29.2 deg; joints [8.952, -65.756, 136.991, 11.786, -75.652, -1.287] of KR 8 1620 ARC HW
    - target stk_p3_s25_t19 (Cartesian target) at (977.09, -132.43, 653.62) mm, rotated rx -27.43 ry 85.45 rz -25.4 deg; joints [8.219, -65.838, 137.112, 10.629, -75.617, -1.305] of KR 8 1620 ARC HW
    - target stk_p3_s25_t20 (Cartesian target) at (977.31, -121.87, 653.74) mm, rotated rx -22.9 ry 85.62 rz -21.25 deg; joints [7.485, -65.913, 137.219, 9.47, -75.584, -1.323] of KR 8 1620 ARC HW
    - target stk_p3_s25_t21 (Cartesian target) at (977.53, -111.31, 653.86) mm, rotated rx -18.04 ry 85.76 rz -16.77 deg; joints [6.748, -65.981, 137.314, 8.308, -75.551, -1.342] of KR 8 1620 ARC HW
    - target stk_p3_s25_t22 (Cartesian target) at (977.75, -100.76, 653.99) mm, rotated rx -12.89 ry 85.87 rz -12 deg; joints [6.01, -66.041, 137.395, 7.144, -75.519, -1.362] of KR 8 1620 ARC HW
    - target stk_p3_s25_t23 (Cartesian target) at (977.97, -90.2, 654.11) mm, rotated rx -7.5 ry 85.94 rz -6.99 deg; joints [5.27, -66.095, 137.463, 5.978, -75.488, -1.381] of KR 8 1620 ARC HW
    - target stk_p3_s25_t24 (Cartesian target) at (978.19, -79.64, 654.23) mm, rotated rx -1.96 ry 85.98 rz -1.83 deg; joints [4.529, -66.141, 137.517, 4.81, -75.458, -1.4] of KR 8 1620 ARC HW
    - target stk_p3_s25_t25 (Cartesian target) at (978.41, -69.08, 654.36) mm, rotated rx 3.62 ry 85.98 rz 3.38 deg; joints [3.787, -66.18, 137.558, 3.641, -75.43, -1.42] of KR 8 1620 ARC HW
    - target stk_p3_s26_t0 (Cartesian target) at (980.06, -20.01, 971.8) mm, rotated rx 165.04 ry 81.99 rz 162.82 deg; joints [0.339, -82.134, 122.335, -3.216, -32.497, 0.397] of KR 8 1620 ARC HW
    - target stk_p3_s26_t0 (Cartesian target) at (980.06, -20.01, 971.8) mm, rotated rx 165.04 ry 81.99 rz 162.82 deg; joints [0.339, -82.134, 122.335, -3.216, -32.497, 0.397] of KR 8 1620 ARC HW
    - target stk_p3_s26_t1 (Cartesian target) at (980.27, -9.45, 971.92) mm, rotated rx 162.39 ry 81.87 rz 159.75 deg; joints [-0.4, -82.117, 122.295, -5.3, -32.536, 1.61] of KR 8 1620 ARC HW
    - target stk_p3_s26_t2 (Cartesian target) at (980.49, 1.11, 972.04) mm, rotated rx 159.81 ry 81.74 rz 156.75 deg; joints [-1.137, -82.089, 122.244, -7.377, -32.604, 2.817] of KR 8 1620 ARC HW
    - target stk_p3_s26_t3 (Cartesian target) at (980.71, 11.67, 972.17) mm, rotated rx 157.33 ry 81.6 rz 153.84 deg; joints [-1.873, -82.052, 122.181, -9.443, -32.702, 4.014] of KR 8 1620 ARC HW
    - target stk_p3_s26_t4 (Cartesian target) at (980.93, 22.23, 972.29) mm, rotated rx 154.93 ry 81.43 rz 151.03 deg; joints [-2.608, -82.005, 122.107, -11.495, -32.83, 5.198] of KR 8 1620 ARC HW
    - target stk_p3_s26_t5 (Cartesian target) at (981.15, 32.79, 972.41) mm, rotated rx 152.62 ry 81.26 rz 148.3 deg; joints [-3.341, -81.948, 122.02, -13.53, -32.986, 6.365] of KR 8 1620 ARC HW
    - target stk_p3_s26_t6 (Cartesian target) at (981.37, 43.34, 972.54) mm, rotated rx 150.41 ry 81.07 rz 145.67 deg; joints [-4.073, -81.881, 121.922, -15.543, -33.17, 7.513] of KR 8 1620 ARC HW
    - target stk_p3_s26_t7 (Cartesian target) at (981.59, 53.9, 972.66) mm, rotated rx 148.29 ry 80.87 rz 143.14 deg; joints [-4.802, -81.804, 121.813, -17.533, -33.381, 8.639] of KR 8 1620 ARC HW
    - target stk_p3_s26_t8 (Cartesian target) at (981.81, 64.46, 972.79) mm, rotated rx 146.27 ry 80.66 rz 140.7 deg; joints [-5.529, -81.718, 121.691, -19.497, -33.619, 9.74] of KR 8 1620 ARC HW
    - target stk_p3_s26_t9 (Cartesian target) at (982.03, 75.02, 972.91) mm, rotated rx 144.34 ry 80.44 rz 138.35 deg; joints [-6.254, -81.621, 121.558, -21.431, -33.883, 10.815] of KR 8 1620 ARC HW
    - target stk_p3_s26_t10 (Cartesian target) at (982.25, 85.58, 973.03) mm, rotated rx 142.51 ry 80.2 rz 136.1 deg; joints [-6.976, -81.515, 121.413, -23.335, -34.172, 11.86] of KR 8 1620 ARC HW
    - target stk_p3_s26_t11 (Cartesian target) at (982.47, 96.14, 973.16) mm, rotated rx 140.76 ry 79.96 rz 133.93 deg; joints [-7.695, -81.399, 121.257, -25.207, -34.485, 12.875] of KR 8 1620 ARC HW
    - target stk_p3_s26_t12 (Cartesian target) at (982.69, 106.69, 973.28) mm, rotated rx 139.09 ry 79.71 rz 131.85 deg; joints [-8.41, -81.274, 121.089, -27.044, -34.821, 13.859] of KR 8 1620 ARC HW
    - target stk_p3_s26_t13 (Cartesian target) at (982.91, 117.25, 973.4) mm, rotated rx 137.51 ry 79.45 rz 129.86 deg; joints [-9.123, -81.139, 120.91, -28.846, -35.179, 14.809] of KR 8 1620 ARC HW
    - target stk_p3_s26_t14 (Cartesian target) at (983.13, 127.81, 973.53) mm, rotated rx 136.01 ry 79.19 rz 127.94 deg; joints [-9.831, -80.995, 120.718, -30.612, -35.557, 15.726] of KR 8 1620 ARC HW
    - target stk_p3_s26_t15 (Cartesian target) at (983.35, 138.37, 973.65) mm, rotated rx 134.58 ry 78.91 rz 126.09 deg; joints [-10.536, -80.842, 120.516, -32.341, -35.955, 16.609] of KR 8 1620 ARC HW
    - target stk_p3_s26_t16 (Cartesian target) at (983.56, 148.93, 973.77) mm, rotated rx 133.22 ry 78.64 rz 124.32 deg; joints [-11.237, -80.68, 120.302, -34.031, -36.372, 17.456] of KR 8 1620 ARC HW
    - target stk_p3_s26_t17 (Cartesian target) at (983.78, 159.49, 973.9) mm, rotated rx 131.92 ry 78.35 rz 122.61 deg; joints [-11.934, -80.508, 120.076, -35.685, -36.807, 18.27] of KR 8 1620 ARC HW
    - target stk_p3_s26_t18 (Cartesian target) at (984, 170.05, 974.02) mm, rotated rx 130.69 ry 78.06 rz 120.97 deg; joints [-12.626, -80.328, 119.839, -37.3, -37.258, 19.048] of KR 8 1620 ARC HW
    - target stk_p3_s26_t19 (Cartesian target) at (984.22, 180.6, 974.14) mm, rotated rx 129.52 ry 77.77 rz 119.39 deg; joints [-13.314, -80.138, 119.59, -38.877, -37.725, 19.792] of KR 8 1620 ARC HW
    - target stk_p3_s26_t20 (Cartesian target) at (984.44, 191.16, 974.27) mm, rotated rx 128.41 ry 77.48 rz 117.87 deg; joints [-13.997, -79.94, 119.33, -40.417, -38.206, 20.502] of KR 8 1620 ARC HW
    - target stk_p3_s26_t21 (Cartesian target) at (984.66, 201.72, 974.39) mm, rotated rx 127.35 ry 77.17 rz 116.4 deg; joints [-14.675, -79.733, 119.058, -41.919, -38.701, 21.178] of KR 8 1620 ARC HW
    - target stk_p3_s26_t22 (Cartesian target) at (984.88, 212.28, 974.51) mm, rotated rx 126.34 ry 76.87 rz 114.98 deg; joints [-15.348, -79.518, 118.776, -43.384, -39.208, 21.822] of KR 8 1620 ARC HW
    - target stk_p3_s26_t23 (Cartesian target) at (985.1, 222.84, 974.64) mm, rotated rx 125.38 ry 76.56 rz 113.61 deg; joints [-16.016, -79.294, 118.481, -44.814, -39.727, 22.433] of KR 8 1620 ARC HW
    - target stk_p3_s26_t24 (Cartesian target) at (985.32, 233.4, 974.76) mm, rotated rx 124.46 ry 76.25 rz 112.28 deg; joints [-16.679, -79.062, 118.175, -46.208, -40.257, 23.013] of KR 8 1620 ARC HW
    - target stk_p3_s26_t25 (Cartesian target) at (985.54, 243.95, 974.89) mm, rotated rx 123.58 ry 75.94 rz 111 deg; joints [-17.336, -78.822, 117.858, -47.567, -40.796, 23.563] of KR 8 1620 ARC HW
    - target stk_p3_s27_t0 (Cartesian target) at (973.48, -336.76, 968.09) mm, rotated rx -128.25 ry 77.87 rz -118.04 deg; joints [21.629, -78.116, 118.026, 49.147, -42.784, -26.234] of KR 8 1620 ARC HW
    - target stk_p3_s27_t0 (Cartesian target) at (973.48, -336.76, 968.09) mm, rotated rx -128.25 ry 77.87 rz -118.04 deg; joints [21.629, -78.116, 118.026, 49.147, -42.784, -26.234] of KR 8 1620 ARC HW
    - target stk_p3_s27_t1 (Cartesian target) at (973.7, -326.2, 968.21) mm, rotated rx -129.42 ry 78.16 rz -119.62 deg; joints [20.977, -78.381, 118.341, 47.884, -42.213, -25.792] of KR 8 1620 ARC HW
    - target stk_p3_s27_t2 (Cartesian target) at (973.91, -315.64, 968.34) mm, rotated rx -130.65 ry 78.44 rz -121.25 deg; joints [20.319, -78.638, 118.643, 46.589, -41.649, -25.322] of KR 8 1620 ARC HW
    - target stk_p3_s27_t3 (Cartesian target) at (974.13, -305.08, 968.46) mm, rotated rx -131.95 ry 78.72 rz -122.96 deg; joints [19.656, -78.886, 118.934, 45.262, -41.093, -24.824] of KR 8 1620 ARC HW
    - target stk_p3_s27_t4 (Cartesian target) at (974.35, -294.53, 968.58) mm, rotated rx -133.31 ry 78.99 rz -124.73 deg; joints [18.988, -79.127, 119.213, 43.901, -40.545, -24.296] of KR 8 1620 ARC HW
    - target stk_p3_s27_t5 (Cartesian target) at (974.57, -283.97, 968.71) mm, rotated rx -134.75 ry 79.26 rz -126.57 deg; joints [18.314, -79.359, 119.481, 42.506, -40.007, -23.738] of KR 8 1620 ARC HW
    - target stk_p3_s27_t6 (Cartesian target) at (974.79, -273.41, 968.83) mm, rotated rx -136.26 ry 79.52 rz -128.49 deg; joints [17.636, -79.582, 119.737, 41.077, -39.48, -23.149] of KR 8 1620 ARC HW
    - target stk_p3_s27_t7 (Cartesian target) at (975.01, -262.85, 968.96) mm, rotated rx -137.84 ry 79.77 rz -130.48 deg; joints [16.953, -79.796, 119.981, 39.611, -38.964, -22.527] of KR 8 1620 ARC HW
    - target stk_p3_s27_t8 (Cartesian target) at (975.23, -252.29, 969.08) mm, rotated rx -139.51 ry 80.02 rz -132.56 deg; joints [16.264, -80.002, 120.213, 38.11, -38.459, -21.872] of KR 8 1620 ARC HW
    - target stk_p3_s27_t9 (Cartesian target) at (975.45, -241.73, 969.2) mm, rotated rx -141.27 ry 80.26 rz -134.73 deg; joints [15.572, -80.199, 120.433, 36.571, -37.969, -21.183] of KR 8 1620 ARC HW
    - target stk_p3_s27_t10 (Cartesian target) at (975.67, -231.17, 969.33) mm, rotated rx -143.11 ry 80.49 rz -136.98 deg; joints [14.875, -80.387, 120.642, 34.996, -37.492, -20.459] of KR 8 1620 ARC HW
    - target stk_p3_s27_t11 (Cartesian target) at (975.89, -220.62, 969.45) mm, rotated rx -145.04 ry 80.71 rz -139.33 deg; joints [14.173, -80.566, 120.839, 33.383, -37.03, -19.701] of KR 8 1620 ARC HW
    - target stk_p3_s27_t12 (Cartesian target) at (976.11, -210.06, 969.57) mm, rotated rx -147.07 ry 80.91 rz -141.77 deg; joints [13.468, -80.736, 121.024, 31.732, -36.585, -18.907] of KR 8 1620 ARC HW
    - target stk_p3_s27_t13 (Cartesian target) at (976.33, -199.5, 969.7) mm, rotated rx -149.19 ry 81.11 rz -144.3 deg; joints [12.759, -80.896, 121.197, 30.044, -36.157, -18.078] of KR 8 1620 ARC HW
    - target stk_p3_s27_t14 (Cartesian target) at (976.55, -188.94, 969.82) mm, rotated rx -151.41 ry 81.3 rz -146.93 deg; joints [12.046, -81.047, 121.359, 28.318, -35.748, -17.214] of KR 8 1620 ARC HW
    - target stk_p3_s27_t15 (Cartesian target) at (976.77, -178.38, 969.94) mm, rotated rx -153.72 ry 81.47 rz -149.66 deg; joints [11.33, -81.188, 121.508, 26.556, -35.358, -16.315] of KR 8 1620 ARC HW
    - target stk_p3_s27_t16 (Cartesian target) at (976.99, -167.82, 970.07) mm, rotated rx -156.12 ry 81.62 rz -152.48 deg; joints [10.611, -81.32, 121.646, 24.757, -34.989, -15.381] of KR 8 1620 ARC HW
    - target stk_p3_s27_t17 (Cartesian target) at (977.2, -157.27, 970.19) mm, rotated rx -158.61 ry 81.77 rz -155.39 deg; joints [9.889, -81.443, 121.772, 22.923, -34.641, -14.414] of KR 8 1620 ARC HW
    - target stk_p3_s27_t18 (Cartesian target) at (977.42, -146.71, 970.31) mm, rotated rx -161.19 ry 81.89 rz -158.39 deg; joints [9.164, -81.556, 121.886, 21.055, -34.316, -13.413] of KR 8 1620 ARC HW
    - target stk_p3_s27_t19 (Cartesian target) at (977.64, -136.15, 970.44) mm, rotated rx -163.85 ry 82 rz -161.46 deg; joints [8.436, -81.658, 121.989, 19.155, -34.015, -12.382] of KR 8 1620 ARC HW
    - target stk_p3_s27_t20 (Cartesian target) at (977.86, -125.59, 970.56) mm, rotated rx -166.58 ry 82.1 rz -164.61 deg; joints [7.706, -81.752, 122.079, 17.223, -33.738, -11.32] of KR 8 1620 ARC HW
    - target stk_p3_s27_t21 (Cartesian target) at (978.08, -115.03, 970.68) mm, rotated rx -169.36 ry 82.17 rz -167.81 deg; joints [6.974, -81.835, 122.158, 15.263, -33.487, -10.231] of KR 8 1620 ARC HW
    - target stk_p3_s27_t22 (Cartesian target) at (978.3, -104.47, 970.81) mm, rotated rx -172.2 ry 82.23 rz -171.06 deg; joints [6.241, -81.908, 122.225, 13.276, -33.263, -9.116] of KR 8 1620 ARC HW
    - target stk_p3_s27_t23 (Cartesian target) at (978.52, -93.92, 970.93) mm, rotated rx -175.07 ry 82.27 rz -174.35 deg; joints [5.506, -81.971, 122.28, 11.266, -33.066, -7.977] of KR 8 1620 ARC HW
    - target stk_p3_s27_t24 (Cartesian target) at (978.74, -83.36, 971.06) mm, rotated rx -177.96 ry 82.28 rz -177.67 deg; joints [4.769, -82.025, 122.323, 9.234, -32.896, -6.818] of KR 8 1620 ARC HW
    - target stk_p3_s27_t25 (Cartesian target) at (978.96, -72.8, 971.18) mm, rotated rx 179.14 ry 82.28 rz 179.02 deg; joints [4.032, -82.068, 122.355, 7.184, -32.756, -5.641] of KR 8 1620 ARC HW
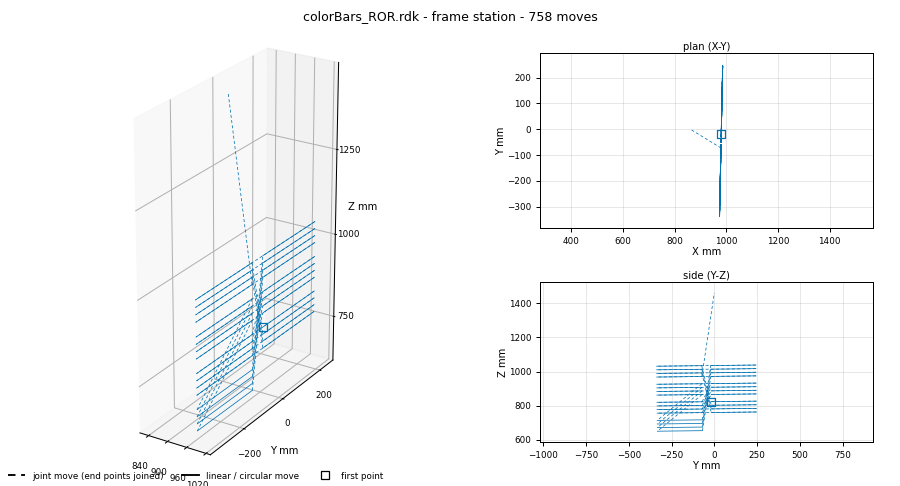
[picture p0: tool path of colorBars_ROR.rdk in frame station, 758 of 758 moves have a stored position in this frame; points joined in program order, loops and branches not executed]

--- program pv_f053_00 (robot KR 8 1620 ARC HW) ---
  Set IO_1=0.0
  Set IO_2=0.0
  Set IO_3=0.0
  Set IO_4=0.0
  Set IO_5=0.0
  Set IO_6=0.0
  Set IO_7=0.0
  Set IO_8=0.0
  Set IO_9=0.0
  Set IO_10=0.0
  Set IO_11=0.0
  Set IO_12=0.0
  Set IO_13=0.0
  Set IO_14=0.0
  Set IO_15=0.0
  Set IO_16=0.0
  Set IO_17=0.0
  Set IO_18=0.0
  Set IO_19=0.0
  Set IO_20=0.0
  Set IO_21=0.0
  Set IO_22=0.0
  Set IO_23=0.0
  Set IO_24=0.0
  Set IO_33=0.0
  Set IO_34=0.0
  Set IO_35=0.0
  Set IO_36=0.0
  MoveJ (init_t0)
  Set IO_49=1.0
  Pause 1.0 s
  Set IO_49=0.0
  Smooth(5)
  Set speed (40.0 mm/s)
  Set speed (15.0 deg/s)
  Set Tool: fbx_2_slot_02_fo3_roundShape_outPaintBrush
  Stroke stk_p0_s0
  Set IO_33=0.0
  Set IO_34=0.0
  Set IO_35=0.0
  Set IO_36=0.0
  MoveJ (stk_p0_s0_t0)
  Set IO_33=0.14000000059604645
  Set IO_35=0.14000000059604645
  MoveL (stk_p0_s0_t0)
  MoveL (stk_p0_s0_t1)
  MoveL (stk_p0_s0_t2)
  MoveL (stk_p0_s0_t3)
  MoveL (stk_p0_s0_t4)
  MoveL (stk_p0_s0_t5)
  MoveL (stk_p0_s0_t6)
  MoveL (stk_p0_s0_t7)
  MoveL (stk_p0_s0_t8)
  MoveL (stk_p0_s0_t9)
  MoveL (stk_p0_s0_t10)
  MoveL (stk_p0_s0_t11)
  MoveL (stk_p0_s0_t12)
  MoveL (stk_p0_s0_t13)
  MoveL (stk_p0_s0_t14)
  MoveL (stk_p0_s0_t15)
  MoveL (stk_p0_s0_t16)
  MoveL (stk_p0_s0_t17)
  MoveL (stk_p0_s0_t18)
  MoveL (stk_p0_s0_t19)
  MoveL (stk_p0_s0_t20)
  MoveL (stk_p0_s0_t21)
  MoveL (stk_p0_s0_t22)
  MoveL (stk_p0_s0_t23)
  MoveL (stk_p0_s0_t24)
  MoveL (stk_p0_s0_t25)
  Set IO_9=0.0
  Set IO_10=0.0
  Set IO_11=0.0
  Set IO_12=0.0
  Set Tool: fbx_2_slot_02_fo3_roundShape_outPaintBrush
  Stroke stk_p0_s1
  Set IO_33=0.0
  Set IO_34=0.0
  Set IO_35=0.0
  Set IO_36=0.0
  MoveJ (stk_p0_s1_t0)
  Set IO_35=0.14000000059604645
  MoveL (stk_p0_s1_t0)
  MoveL (stk_p0_s1_t1)
  MoveL (stk_p0_s1_t2)
  MoveL (stk_p0_s1_t3)
  MoveL (stk_p0_s1_t4)
  MoveL (stk_p0_s1_t5)
  MoveL (stk_p0_s1_t6)
  MoveL (stk_p0_s1_t7)
  MoveL (stk_p0_s1_t8)
  MoveL (stk_p0_s1_t9)
  MoveL (stk_p0_s1_t10)
  MoveL (stk_p0_s1_t11)
  MoveL (stk_p0_s1_t12)
  MoveL (stk_p0_s1_t13)
  MoveL (stk_p0_s1_t14)
  MoveL (stk_p0_s1_t15)
  MoveL (stk_p0_s1_t16)
  MoveL (stk_p0_s1_t17)
  MoveL (stk_p0_s1_t18)
  MoveL (stk_p0_s1_t19)
  MoveL (stk_p0_s1_t20)
  MoveL (stk_p0_s1_t21)
  MoveL (stk_p0_s1_t22)
  MoveL (stk_p0_s1_t23)
  MoveL (stk_p0_s1_t24)
  MoveL (stk_p0_s1_t25)
  Set IO_9=0.0
  Set IO_10=0.0
  Set IO_11=0.0
  Set IO_12=0.0
  Set Tool: fbx_2_slot_02_fo3_roundShape_outPaintBrush
  Stroke stk_p0_s2
  Set IO_33=0.0
  Set IO_34=0.0
  Set IO_35=0.0
  Set IO_36=0.0
  MoveJ (stk_p0_s2_t0)
  Set IO_34=0.14000000059604645
  Set IO_35=0.14000000059604645
  MoveL (stk_p0_s2_t0)
  MoveL (stk_p0_s2_t1)
  MoveL (stk_p0_s2_t2)
  MoveL (stk_p0_s2_t3)
  MoveL (stk_p0_s2_t4)
  MoveL (stk_p0_s2_t5)
  MoveL (stk_p0_s2_t6)
  MoveL (stk_p0_s2_t7)
  MoveL (stk_p0_s2_t8)
  MoveL (stk_p0_s2_t9)
  MoveL (stk_p0_s2_t10)
  MoveL (stk_p0_s2_t11)
  MoveL (stk_p0_s2_t12)
  MoveL (stk_p0_s2_t13)
  MoveL (stk_p0_s2_t14)
  MoveL (stk_p0_s2_t15)
  MoveL (stk_p0_s2_t16)
  MoveL (stk_p0_s2_t17)
  MoveL (stk_p0_s2_t18)
  MoveL (stk_p0_s2_t19)
  MoveL (stk_p0_s2_t20)
  MoveL (stk_p0_s2_t21)
  MoveL (stk_p0_s2_t22)
  MoveL (stk_p0_s2_t23)
  MoveL (stk_p0_s2_t24)
  MoveL (stk_p0_s2_t25)
  Set IO_9=0.0
  Set IO_10=0.0
  Set IO_11=0.0
  Set IO_12=0.0
  Set Tool: fbx_2_slot_02_fo3_roundShape_outPaintBrush
  Stroke stk_p0_s3
  Set IO_33=0.0
  Set IO_34=0.0
  Set IO_35=0.0
  Set IO_36=0.0
  MoveJ (stk_p0_s3_t0)
  Set IO_34=0.14000000059604645
  MoveL (stk_p0_s3_t0)
  MoveL (stk_p0_s3_t1)
  MoveL (stk_p0_s3_t2)
  MoveL (stk_p0_s3_t3)
  MoveL (stk_p0_s3_t4)
  MoveL (stk_p0_s3_t5)
  MoveL (stk_p0_s3_t6)
  MoveL (stk_p0_s3_t7)
  MoveL (stk_p0_s3_t8)
  MoveL (stk_p0_s3_t9)
  MoveL (stk_p0_s3_t10)
  MoveL (stk_p0_s3_t11)
  MoveL (stk_p0_s3_t12)
  MoveL (stk_p0_s3_t13)
  MoveL (stk_p0_s3_t14)
  MoveL (stk_p0_s3_t15)
  MoveL (stk_p0_s3_t16)
  MoveL (stk_p0_s3_t17)
  MoveL (stk_p0_s3_t18)
  MoveL (stk_p0_s3_t19)
  MoveL (stk_p0_s3_t20)
  MoveL (stk_p0_s3_t21)
  MoveL (stk_p0_s3_t22)
  MoveL (stk_p0_s3_t23)
  MoveL (stk_p0_s3_t24)
  MoveL (stk_p0_s3_t25)
  Set IO_9=0.0
  Set IO_10=0.0
  Set IO_11=0.0
  Set IO_12=0.0
  Set Tool: fbx_2_slot_02_fo3_roundShape_outPaintBrush
  Stroke stk_p0_s4
  Set IO_33=0.0
  Set IO_34=0.0
  Set IO_35=0.0
  Set IO_36=0.0
  MoveJ (stk_p0_s4_t0)
  Set IO_33=0.14000000059604645
  Set IO_34=0.14000000059604645
  Set IO_35=0.14000000059604645
  MoveL (stk_p0_s4_t0)
  MoveL (stk_p0_s4_t1)
  MoveL (stk_p0_s4_t2)
  MoveL (stk_p0_s4_t3)
  MoveL (stk_p0_s4_t4)
  MoveL (stk_p0_s4_t5)
  MoveL (stk_p0_s4_t6)
  MoveL (stk_p0_s4_t7)
  MoveL (stk_p0_s4_t8)
  MoveL (stk_p0_s4_t9)
  MoveL (stk_p0_s4_t10)
  MoveL (stk_p0_s4_t11)
  MoveL (stk_p0_s4_t12)
  MoveL (stk_p0_s4_t13)
  MoveL (stk_p0_s4_t14)
  MoveL (stk_p0_s4_t15)
  MoveL (stk_p0_s4_t16)
  MoveL (stk_p0_s4_t17)
  MoveL (stk_p0_s4_t18)
  MoveL (stk_p0_s4_t19)
  MoveL (stk_p0_s4_t20)
  MoveL (stk_p0_s4_t21)
  MoveL (stk_p0_s4_t22)
  MoveL (stk_p0_s4_t23)
  MoveL (stk_p0_s4_t24)
  MoveL (stk_p0_s4_t25)
  Set IO_9=0.0
  Set IO_10=0.0
  Set IO_11=0.0
  Set IO_12=0.0
  Set Tool: fbx_2_slot_02_fo3_roundShape_outPaintBrush
  Stroke stk_p0_s5
  Set IO_33=0.0
  Set IO_34=0.0
  Set IO_35=0.0
  Set IO_36=0.0
  MoveJ (stk_p0_s5_t0)
  Set IO_33=0.14000000059604645
  Set IO_34=0.14000000059604645
  MoveL (stk_p0_s5_t0)
  MoveL (stk_p0_s5_t1)
  MoveL (stk_p0_s5_t2)
  MoveL (stk_p0_s5_t3)
  MoveL (stk_p0_s5_t4)
  MoveL (stk_p0_s5_t5)
  MoveL (stk_p0_s5_t6)
  MoveL (stk_p0_s5_t7)
  MoveL (stk_p0_s5_t8)
  MoveL (stk_p0_s5_t9)
  MoveL (stk_p0_s5_t10)
  MoveL (stk_p0_s5_t11)
  MoveL (stk_p0_s5_t12)
  MoveL (stk_p0_s5_t13)
  MoveL (stk_p0_s5_t14)
  MoveL (stk_p0_s5_t15)
  MoveL (stk_p0_s5_t16)
  MoveL (stk_p0_s5_t17)
  MoveL (stk_p0_s5_t18)
  MoveL (stk_p0_s5_t19)
  MoveL (stk_p0_s5_t20)
  MoveL (stk_p0_s5_t21)
  MoveL (stk_p0_s5_t22)
  MoveL (stk_p0_s5_t23)
  MoveL (stk_p0_s5_t24)
  MoveL (stk_p0_s5_t25)
  Set IO_9=0.0
  Set IO_10=0.0
  Set IO_11=0.0
  Set IO_12=0.0
  Set Tool: fbx_2_slot_02_fo3_roundShape_outPaintBrush
  Stroke stk_p0_s6
  Set IO_33=0.0
  Set IO_34=0.0
  Set IO_35=0.0
  Set IO_36=0.0
  MoveJ (stk_p0_s6_t0)
  Set IO_33=0.14000000059604645
  MoveL (stk_p0_s6_t0)
  MoveL (stk_p0_s6_t1)
  MoveL (stk_p0_s6_t2)
  MoveL (stk_p0_s6_t3)
  MoveL (stk_p0_s6_t4)
  MoveL (stk_p0_s6_t5)
  MoveL (stk_p0_s6_t6)
  MoveL (stk_p0_s6_t7)
  MoveL (stk_p0_s6_t8)
  MoveL (stk_p0_s6_t9)
  MoveL (stk_p0_s6_t10)
  MoveL (stk_p0_s6_t11)
  MoveL (stk_p0_s6_t12)
  MoveL (stk_p0_s6_t13)
  MoveL (stk_p0_s6_t14)
  MoveL (stk_p0_s6_t15)
  MoveL (stk_p0_s6_t16)
  MoveL (stk_p0_s6_t17)
  MoveL (stk_p0_s6_t18)
  MoveL (stk_p0_s6_t19)
  MoveL (stk_p0_s6_t20)
  MoveL (stk_p0_s6_t21)
  MoveL (stk_p0_s6_t22)
  MoveL (stk_p0_s6_t23)
  MoveL (stk_p0_s6_t24)
  MoveL (stk_p0_s6_t25)
  Set IO_9=0.0
  Set IO_10=0.0
  Set IO_11=0.0
  Set IO_12=0.0
  Set Tool: fbx_3_slot_03_fo4_roundShape_outPaintBrush
  Stroke stk_p1_s7
  Set IO_37=0.0
  Set IO_38=0.0
  Set IO_39=0.0
  Set IO_40=0.0
  MoveJ (stk_p1_s7_t0)
  Set IO_37=0.14000000059604645
  Set IO_39=0.14000000059604645
  MoveL (stk_p1_s7_t0)
  MoveL (stk_p1_s7_t1)
  MoveL (stk_p1_s7_t2)
  MoveL (stk_p1_s7_t3)
  MoveL (stk_p1_s7_t4)
  MoveL (stk_p1_s7_t5)
  MoveL (stk_p1_s7_t6)
  MoveL (stk_p1_s7_t7)
  MoveL (stk_p1_s7_t8)
  MoveL (stk_p1_s7_t9)
  MoveL (stk_p1_s7_t10)
  MoveL (stk_p1_s7_t11)
  MoveL (stk_p1_s7_t12)
  MoveL (stk_p1_s7_t13)
  MoveL (stk_p1_s7_t14)
  MoveL (stk_p1_s7_t15)
  MoveL (stk_p1_s7_t16)
  MoveL (stk_p1_s7_t17)
  MoveL (stk_p1_s7_t18)
  MoveL (stk_p1_s7_t19)
  MoveL (stk_p1_s7_t20)
  MoveL (stk_p1_s7_t21)
  MoveL (stk_p1_s7_t22)
  MoveL (stk_p1_s7_t23)
  MoveL (stk_p1_s7_t24)
  MoveL (stk_p1_s7_t25)
  Set IO_13=0.0
  Set IO_14=0.0
  Set IO_15=0.0
  Set IO_16=0.0
  Set Tool: fbx_3_slot_03_fo4_roundShape_outPaintBrush
  Stroke stk_p1_s8
  Set IO_37=0.0
  Set IO_38=0.0
  Set IO_39=0.0
  Set IO_40=0.0
  MoveJ (stk_p1_s8_t0)
  Set IO_39=0.14000000059604645
  MoveL (stk_p1_s8_t0)
  MoveL (stk_p1_s8_t1)
  MoveL (stk_p1_s8_t2)
  MoveL (stk_p1_s8_t3)
  MoveL (stk_p1_s8_t4)
  MoveL (stk_p1_s8_t5)
  MoveL (stk_p1_s8_t6)
  MoveL (stk_p1_s8_t7)
  MoveL (stk_p1_s8_t8)
  MoveL (stk_p1_s8_t9)
  MoveL (stk_p1_s8_t10)
  MoveL (stk_p1_s8_t11)
  MoveL (stk_p1_s8_t12)
  MoveL (stk_p1_s8_t13)
  MoveL (stk_p1_s8_t14)
  MoveL (stk_p1_s8_t15)
  MoveL (stk_p1_s8_t16)
  MoveL (stk_p1_s8_t17)
  MoveL (stk_p1_s8_t18)
  MoveL (stk_p1_s8_t19)
  MoveL (stk_p1_s8_t20)
  MoveL (stk_p1_s8_t21)
  MoveL (stk_p1_s8_t22)
  MoveL (stk_p1_s8_t23)
  MoveL (stk_p1_s8_t24)
  MoveL (stk_p1_s8_t25)
  Set IO_13=0.0
  Set IO_14=0.0
  Set IO_15=0.0
  Set IO_16=0.0
  Set Tool: fbx_3_slot_03_fo4_roundShape_outPaintBrush
  Stroke stk_p1_s9
  Set IO_37=0.0
  Set IO_38=0.0
  Set IO_39=0.0
  Set IO_40=0.0
  MoveJ (stk_p1_s9_t0)
  Set IO_38=0.14000000059604645
  Set IO_39=0.14000000059604645
  MoveL (stk_p1_s9_t0)
  MoveL (stk_p1_s9_t1)
  MoveL (stk_p1_s9_t2)
  MoveL (stk_p1_s9_t3)
  MoveL (stk_p1_s9_t4)
  MoveL (stk_p1_s9_t5)
  MoveL (stk_p1_s9_t6)
  MoveL (stk_p1_s9_t7)
  MoveL (stk_p1_s9_t8)
  MoveL (stk_p1_s9_t9)
  MoveL (stk_p1_s9_t10)
  MoveL (stk_p1_s9_t11)
  MoveL (stk_p1_s9_t12)
  MoveL (stk_p1_s9_t13)
  MoveL (stk_p1_s9_t14)
  MoveL (stk_p1_s9_t15)
  MoveL (stk_p1_s9_t16)
  MoveL (stk_p1_s9_t17)
  MoveL (stk_p1_s9_t18)
  MoveL (stk_p1_s9_t19)
  MoveL (stk_p1_s9_t20)
  MoveL (stk_p1_s9_t21)
  MoveL (stk_p1_s9_t22)
  MoveL (stk_p1_s9_t23)
  MoveL (stk_p1_s9_t24)
  MoveL (stk_p1_s9_t25)
  Set IO_13=0.0
  Set IO_14=0.0
  Set IO_15=0.0
  Set IO_16=0.0
  Set Tool: fbx_3_slot_03_fo4_roundShape_outPaintBrush
  Stroke stk_p1_s10
  Set IO_37=0.0
  Set IO_38=0.0
  Set IO_39=0.0
  Set IO_40=0.0
  MoveJ (stk_p1_s10_t0)
  Set IO_38=0.14000000059604645
  MoveL (stk_p1_s10_t0)
  MoveL (stk_p1_s10_t1)
  MoveL (stk_p1_s10_t2)
  MoveL (stk_p1_s10_t3)
  MoveL (stk_p1_s10_t4)
  MoveL (stk_p1_s10_t5)
  MoveL (stk_p1_s10_t6)
  MoveL (stk_p1_s10_t7)
  MoveL (stk_p1_s10_t8)
  MoveL (stk_p1_s10_t9)
  MoveL (stk_p1_s10_t10)
  MoveL (stk_p1_s10_t11)
  MoveL (stk_p1_s10_t12)
  MoveL (stk_p1_s10_t13)
  MoveL (stk_p1_s10_t14)
  MoveL (stk_p1_s10_t15)
  MoveL (stk_p1_s10_t16)
  MoveL (stk_p1_s10_t17)
  MoveL (stk_p1_s10_t18)
  MoveL (stk_p1_s10_t19)
  MoveL (stk_p1_s10_t20)
  MoveL (stk_p1_s10_t21)
  MoveL (stk_p1_s10_t22)
  MoveL (stk_p1_s10_t23)
  MoveL (stk_p1_s10_t24)
  MoveL (stk_p1_s10_t25)
  Set IO_13=0.0
  Set IO_14=0.0
  Set IO_15=0.0
  Set IO_16=0.0
  Set Tool: fbx_3_slot_03_fo4_roundShape_outPaintBrush
  Stroke stk_p1_s11
  Set IO_37=0.0
  Set IO_38=0.0
  Set IO_39=0.0
  Set IO_40=0.0
  MoveJ (stk_p1_s11_t0)
  Set IO_37=0.14000000059604645
  Set IO_38=0.14000000059604645
  Set IO_39=0.14000000059604645
  MoveL (stk_p1_s11_t0)
  MoveL (stk_p1_s11_t1)
  MoveL (stk_p1_s11_t2)
  MoveL (stk_p1_s11_t3)
  MoveL (stk_p1_s11_t4)
  MoveL (stk_p1_s11_t5)
  MoveL (stk_p1_s11_t6)
  MoveL (stk_p1_s11_t7)
  MoveL (stk_p1_s11_t8)
  MoveL (stk_p1_s11_t9)
  MoveL (stk_p1_s11_t10)
  MoveL (stk_p1_s11_t11)
  MoveL (stk_p1_s11_t12)
  MoveL (stk_p1_s11_t13)
  MoveL (stk_p1_s11_t14)
  MoveL (stk_p1_s11_t15)
  MoveL (stk_p1_s11_t16)
  MoveL (stk_p1_s11_t17)
  MoveL (stk_p1_s11_t18)
  MoveL (stk_p1_s11_t19)
  MoveL (stk_p1_s11_t20)
  MoveL (stk_p1_s11_t21)
  MoveL (stk_p1_s11_t22)
  MoveL (stk_p1_s11_t23)
  MoveL (stk_p1_s11_t24)
  MoveL (stk_p1_s11_t25)
  Set IO_13=0.0
  Set IO_14=0.0
  Set IO_15=0.0
  Set IO_16=0.0
  Set Tool: fbx_3_slot_03_fo4_roundShape_outPaintBrush
  Stroke stk_p1_s12
  Set IO_37=0.0
  Set IO_38=0.0
  Set IO_39=0.0
  Set IO_40=0.0
  MoveJ (stk_p1_s12_t0)
  Set IO_37=0.14000000059604645
  Set IO_38=0.14000000059604645
  MoveL (stk_p1_s12_t0)
  MoveL (stk_p1_s12_t1)
  MoveL (stk_p1_s12_t2)
  MoveL (stk_p1_s12_t3)
  MoveL (stk_p1_s12_t4)
  MoveL (stk_p1_s12_t5)
  MoveL (stk_p1_s12_t6)
  MoveL (stk_p1_s12_t7)
  MoveL (stk_p1_s12_t8)
  MoveL (stk_p1_s12_t9)
  MoveL (stk_p1_s12_t10)
  MoveL (stk_p1_s12_t11)
  MoveL (stk_p1_s12_t12)
  MoveL (stk_p1_s12_t13)
  MoveL (stk_p1_s12_t14)
  MoveL (stk_p1_s12_t15)
  MoveL (stk_p1_s12_t16)
  MoveL (stk_p1_s12_t17)
  MoveL (stk_p1_s12_t18)
  MoveL (stk_p1_s12_t19)
  MoveL (stk_p1_s12_t20)
  MoveL (stk_p1_s12_t21)
  MoveL (stk_p1_s12_t22)
  MoveL (stk_p1_s12_t23)
  MoveL (stk_p1_s12_t24)
  MoveL (stk_p1_s12_t25)
  Set IO_13=0.0
  Set IO_14=0.0
  Set IO_15=0.0
  Set IO_16=0.0
  Set Tool: fbx_3_slot_03_fo4_roundShape_outPaintBrush
  Stroke stk_p1_s13
  Set IO_37=0.0
  Set IO_38=0.0
  Set IO_39=0.0
  Set IO_40=0.0
  MoveJ (stk_p1_s13_t0)
  Set IO_37=0.14000000059604645
  MoveL (stk_p1_s13_t0)
  MoveL (stk_p1_s13_t1)
  MoveL (stk_p1_s13_t2)
  MoveL (stk_p1_s13_t3)
  MoveL (stk_p1_s13_t4)
  MoveL (stk_p1_s13_t5)
  MoveL (stk_p1_s13_t6)
  MoveL (stk_p1_s13_t7)
  MoveL (stk_p1_s13_t8)
  MoveL (stk_p1_s13_t9)
  MoveL (stk_p1_s13_t10)
  MoveL (stk_p1_s13_t11)
  MoveL (stk_p1_s13_t12)
  MoveL (stk_p1_s13_t13)
  MoveL (stk_p1_s13_t14)
  MoveL (stk_p1_s13_t15)
  MoveL (stk_p1_s13_t16)
  MoveL (stk_p1_s13_t17)
  MoveL (stk_p1_s13_t18)
  MoveL (stk_p1_s13_t19)
  MoveL (stk_p1_s13_t20)
  MoveL (stk_p1_s13_t21)
  MoveL (stk_p1_s13_t22)
  MoveL (stk_p1_s13_t23)
  MoveL (stk_p1_s13_t24)
  MoveL (stk_p1_s13_t25)
  Set IO_13=0.0
  Set IO_14=0.0
  Set IO_15=0.0
  Set IO_16=0.0
  Set Tool: fbx_4_slot_04_fo5_roundShape_outPaintBrush
  Stroke stk_p2_s14
  Set IO_41=0.0
  Set IO_42=0.0
  Set IO_43=0.0
  Set IO_44=0.0
  MoveJ (stk_p2_s14_t0)
  Set IO_41=0.14000000059604645
  Set IO_43=0.14000000059604645
  MoveL (stk_p2_s14_t0)
  MoveL (stk_p2_s14_t1)
  MoveL (stk_p2_s14_t2)
  MoveL (stk_p2_s14_t3)
  MoveL (stk_p2_s14_t4)
  MoveL (stk_p2_s14_t5)
  MoveL (stk_p2_s14_t6)
  MoveL (stk_p2_s14_t7)
  MoveL (stk_p2_s14_t8)
  MoveL (stk_p2_s14_t9)
  MoveL (stk_p2_s14_t10)
  MoveL (stk_p2_s14_t11)
  MoveL (stk_p2_s14_t12)
  MoveL (stk_p2_s14_t13)
  MoveL (stk_p2_s14_t14)
  MoveL (stk_p2_s14_t15)
  MoveL (stk_p2_s14_t16)
  MoveL (stk_p2_s14_t17)
  MoveL (stk_p2_s14_t18)
  MoveL (stk_p2_s14_t19)
  MoveL (stk_p2_s14_t20)
  MoveL (stk_p2_s14_t21)
  MoveL (stk_p2_s14_t22)
  MoveL (stk_p2_s14_t23)
  MoveL (stk_p2_s14_t24)
  MoveL (stk_p2_s14_t25)
  Set IO_17=0.0
  Set IO_18=0.0
  Set IO_19=0.0
  Set IO_20=0.0
  Set Tool: fbx_4_slot_04_fo5_roundShape_outPaintBrush
  Stroke stk_p2_s15
  Set IO_41=0.0
  Set IO_42=0.0
  Set IO_43=0.0
  Set IO_44=0.0
  MoveJ (stk_p2_s15_t0)
  Set IO_43=0.14000000059604645
  MoveL (stk_p2_s15_t0)
  MoveL (stk_p2_s15_t1)
  MoveL (stk_p2_s15_t2)
  MoveL (stk_p2_s15_t3)
  MoveL (stk_p2_s15_t4)
  MoveL (stk_p2_s15_t5)
  MoveL (stk_p2_s15_t6)
  MoveL (stk_p2_s15_t7)
  MoveL (stk_p2_s15_t8)
  MoveL (stk_p2_s15_t9)
  MoveL (stk_p2_s15_t10)
  MoveL (stk_p2_s15_t11)
  MoveL (stk_p2_s15_t12)
  MoveL (stk_p2_s15_t13)
  MoveL (stk_p2_s15_t14)
  MoveL (stk_p2_s15_t15)
  MoveL (stk_p2_s15_t16)
  MoveL (stk_p2_s15_t17)
  MoveL (stk_p2_s15_t18)
  MoveL (stk_p2_s15_t19)
  MoveL (stk_p2_s15_t20)
  MoveL (stk_p2_s15_t21)
  MoveL (stk_p2_s15_t22)
  MoveL (stk_p2_s15_t23)
  MoveL (stk_p2_s15_t24)
  MoveL (stk_p2_s15_t25)
  Set IO_17=0.0
  Set IO_18=0.0
  Set IO_19=0.0
  Set IO_20=0.0
  Set Tool: fbx_4_slot_04_fo5_roundShape_outPaintBrush
  Stroke stk_p2_s16
  Set IO_41=0.0
  Set IO_42=0.0
  Set IO_43=0.0
  Set IO_44=0.0
  MoveJ (stk_p2_s16_t0)
  Set IO_42=0.14000000059604645
  Set IO_43=0.14000000059604645
  MoveL (stk_p2_s16_t0)
  MoveL (stk_p2_s16_t1)
  MoveL (stk_p2_s16_t2)
  MoveL (stk_p2_s16_t3)
  MoveL (stk_p2_s16_t4)
  MoveL (stk_p2_s16_t5)
  MoveL (stk_p2_s16_t6)
  MoveL (stk_p2_s16_t7)
  MoveL (stk_p2_s16_t8)
  MoveL (stk_p2_s16_t9)
  MoveL (stk_p2_s16_t10)
  MoveL (stk_p2_s16_t11)
  MoveL (stk_p2_s16_t12)
  MoveL (stk_p2_s16_t13)
  MoveL (stk_p2_s16_t14)
  MoveL (stk_p2_s16_t15)
  MoveL (stk_p2_s16_t16)
  MoveL (stk_p2_s16_t17)
  MoveL (stk_p2_s16_t18)
  MoveL (stk_p2_s16_t19)
  MoveL (stk_p2_s16_t20)
  MoveL (stk_p2_s16_t21)
  MoveL (stk_p2_s16_t22)
  MoveL (stk_p2_s16_t23)
  MoveL (stk_p2_s16_t24)
  MoveL (stk_p2_s16_t25)
  Set IO_17=0.0
  Set IO_18=0.0
  Set IO_19=0.0
  Set IO_20=0.0
  Set Tool: fbx_4_slot_04_fo5_roundShape_outPaintBrush
  Stroke stk_p2_s17
  Set IO_41=0.0
  Set IO_42=0.0
  Set IO_43=0.0
  Set IO_44=0.0
  MoveJ (stk_p2_s17_t0)
  Set IO_42=0.14000000059604645
  MoveL (stk_p2_s17_t0)
  MoveL (stk_p2_s17_t1)
  MoveL (stk_p2_s17_t2)
  MoveL (stk_p2_s17_t3)
  MoveL (stk_p2_s17_t4)
  MoveL (stk_p2_s17_t5)
  MoveL (stk_p2_s17_t6)
  MoveL (stk_p2_s17_t7)
  MoveL (stk_p2_s17_t8)
  MoveL (stk_p2_s17_t9)
  MoveL (stk_p2_s17_t10)
  MoveL (stk_p2_s17_t11)
  MoveL (stk_p2_s17_t12)
  MoveL (stk_p2_s17_t13)
  MoveL (stk_p2_s17_t14)
  MoveL (stk_p2_s17_t15)
  MoveL (stk_p2_s17_t16)
  MoveL (stk_p2_s17_t17)
  MoveL (stk_p2_s17_t18)
  MoveL (stk_p2_s17_t19)
  MoveL (stk_p2_s17_t20)
  MoveL (stk_p2_s17_t21)
  MoveL (stk_p2_s17_t22)
  MoveL (stk_p2_s17_t23)
  MoveL (stk_p2_s17_t24)
  MoveL (stk_p2_s17_t25)
  Set IO_17=0.0
  Set IO_18=0.0
  Set IO_19=0.0
  Set IO_20=0.0
  Set Tool: fbx_4_slot_04_fo5_roundShape_outPaintBrush
  Stroke stk_p2_s18
  Set IO_41=0.0
  Set IO_42=0.0
  Set IO_43=0.0
  Set IO_44=0.0
  MoveJ (stk_p2_s18_t0)
  Set IO_41=0.14000000059604645
  Set IO_42=0.14000000059604645
  Set IO_43=0.14000000059604645
  MoveL (stk_p2_s18_t0)
  MoveL (stk_p2_s18_t1)
  MoveL (stk_p2_s18_t2)
  MoveL (stk_p2_s18_t3)
  MoveL (stk_p2_s18_t4)
  MoveL (stk_p2_s18_t5)
  MoveL (stk_p2_s18_t6)
  MoveL (stk_p2_s18_t7)
  MoveL (stk_p2_s18_t8)
  MoveL (stk_p2_s18_t9)
  MoveL (stk_p2_s18_t10)
  MoveL (stk_p2_s18_t11)
  MoveL (stk_p2_s18_t12)
  MoveL (stk_p2_s18_t13)
  MoveL (stk_p2_s18_t14)
  MoveL (stk_p2_s18_t15)
  MoveL (stk_p2_s18_t16)
  MoveL (stk_p2_s18_t17)
  MoveL (stk_p2_s18_t18)
  MoveL (stk_p2_s18_t19)
  MoveL (stk_p2_s18_t20)
  MoveL (stk_p2_s18_t21)
  MoveL (stk_p2_s18_t22)
  MoveL (stk_p2_s18_t23)
  MoveL (stk_p2_s18_t24)
  MoveL (stk_p2_s18_t25)
  Set IO_17=0.0
  Set IO_18=0.0
  Set IO_19=0.0
  Set IO_20=0.0
  Set Tool: fbx_4_slot_04_fo5_roundShape_outPaintBrush
  Stroke stk_p2_s19
  Set IO_41=0.0
  Set IO_42=0.0
  Set IO_43=0.0
  Set IO_44=0.0
  MoveJ (stk_p2_s19_t0)
  Set IO_41=0.14000000059604645
  Set IO_42=0.14000000059604645
  MoveL (stk_p2_s19_t0)
  MoveL (stk_p2_s19_t1)
  MoveL (stk_p2_s19_t2)
  MoveL (stk_p2_s19_t3)
  MoveL (stk_p2_s19_t4)
  MoveL (stk_p2_s19_t5)
  MoveL (stk_p2_s19_t6)
  MoveL (stk_p2_s19_t7)
  MoveL (stk_p2_s19_t8)
  MoveL (stk_p2_s19_t9)
  MoveL (stk_p2_s19_t10)
  MoveL (stk_p2_s19_t11)
  MoveL (stk_p2_s19_t12)
  MoveL (stk_p2_s19_t13)
  MoveL (stk_p2_s19_t14)
  MoveL (stk_p2_s19_t15)
  MoveL (stk_p2_s19_t16)
  MoveL (stk_p2_s19_t17)
  MoveL (stk_p2_s19_t18)
  MoveL (stk_p2_s19_t19)
  MoveL (stk_p2_s19_t20)
  MoveL (stk_p2_s19_t21)
  MoveL (stk_p2_s19_t22)
  MoveL (stk_p2_s19_t23)
  MoveL (stk_p2_s19_t24)
  MoveL (stk_p2_s19_t25)
  Set IO_17=0.0
  Set IO_18=0.0
  Set IO_19=0.0
  Set IO_20=0.0
  Set Tool: fbx_4_slot_04_fo5_roundShape_outPaintBrush
  Stroke stk_p2_s20
  Set IO_41=0.0
  Set IO_42=0.0
  Set IO_43=0.0
  Set IO_44=0.0
  MoveJ (stk_p2_s20_t0)
  Set IO_41=0.14000000059604645
  MoveL (stk_p2_s20_t0)
  MoveL (stk_p2_s20_t1)
  MoveL (stk_p2_s20_t2)
  MoveL (stk_p2_s20_t3)
  MoveL (stk_p2_s20_t4)
  MoveL (stk_p2_s20_t5)
  MoveL (stk_p2_s20_t6)
  MoveL (stk_p2_s20_t7)
  MoveL (stk_p2_s20_t8)
  MoveL (stk_p2_s20_t9)
  MoveL (stk_p2_s20_t10)
  MoveL (stk_p2_s20_t11)
  MoveL (stk_p2_s20_t12)
  MoveL (stk_p2_s20_t13)
  MoveL (stk_p2_s20_t14)
  MoveL (stk_p2_s20_t15)
  MoveL (stk_p2_s20_t16)
  MoveL (stk_p2_s20_t17)
  MoveL (stk_p2_s20_t18)
  MoveL (stk_p2_s20_t19)
  MoveL (stk_p2_s20_t20)
  MoveL (stk_p2_s20_t21)
  MoveL (stk_p2_s20_t22)
  MoveL (stk_p2_s20_t23)
  MoveL (stk_p2_s20_t24)
  MoveL (stk_p2_s20_t25)
  Set IO_17=0.0
  Set IO_18=0.0
  Set IO_19=0.0
  Set IO_20=0.0
  Set Tool: fbx_5_slot_05_fo6_roundShape_outPaintBrush
  Stroke stk_p3_s21
  Set IO_45=0.0
  Set IO_46=0.0
  Set IO_47=0.0
  Set IO_48=0.0
  MoveJ (stk_p3_s21_t0)
  Set IO_45=0.14000000059604645
  Set IO_47=0.14000000059604645
  MoveL (stk_p3_s21_t0)
  MoveL (stk_p3_s21_t1)
  MoveL (stk_p3_s21_t2)
  MoveL (stk_p3_s21_t3)
  MoveL (stk_p3_s21_t4)
  MoveL (stk_p3_s21_t5)
  MoveL (stk_p3_s21_t6)
  MoveL (stk_p3_s21_t7)
  MoveL (stk_p3_s21_t8)
  MoveL (stk_p3_s21_t9)
  MoveL (stk_p3_s21_t10)
  MoveL (stk_p3_s21_t11)
  MoveL (stk_p3_s21_t12)
  MoveL (stk_p3_s21_t13)
  MoveL (stk_p3_s21_t14)
  MoveL (stk_p3_s21_t15)
  MoveL (stk_p3_s21_t16)
  MoveL (stk_p3_s21_t17)
  MoveL (stk_p3_s21_t18)
  MoveL (stk_p3_s21_t19)
  MoveL (stk_p3_s21_t20)
  MoveL (stk_p3_s21_t21)
  MoveL (stk_p3_s21_t22)
  MoveL (stk_p3_s21_t23)
  MoveL (stk_p3_s21_t24)
  MoveL (stk_p3_s21_t25)
  Set IO_21=0.0
  Set IO_22=0.0
  Set IO_23=0.0
  Set IO_24=0.0
  Set Tool: fbx_5_slot_05_fo6_roundShape_outPaintBrush
  Stroke stk_p3_s22
  Set IO_45=0.0
  Set IO_46=0.0
  Set IO_47=0.0
  Set IO_48=0.0
  MoveJ (stk_p3_s22_t0)
  Set IO_47=0.14000000059604645
  MoveL (stk_p3_s22_t0)
  MoveL (stk_p3_s22_t1)
  MoveL (stk_p3_s22_t2)
  MoveL (stk_p3_s22_t3)
  MoveL (stk_p3_s22_t4)
  MoveL (stk_p3_s22_t5)
  MoveL (stk_p3_s22_t6)
  MoveL (stk_p3_s22_t7)
  MoveL (stk_p3_s22_t8)
  MoveL (stk_p3_s22_t9)
  MoveL (stk_p3_s22_t10)
  MoveL (stk_p3_s22_t11)
  MoveL (stk_p3_s22_t12)
  MoveL (stk_p3_s22_t13)
  MoveL (stk_p3_s22_t14)
  MoveL (stk_p3_s22_t15)
  MoveL (stk_p3_s22_t16)
  MoveL (stk_p3_s22_t17)
  MoveL (stk_p3_s22_t18)
  MoveL (stk_p3_s22_t19)
  MoveL (stk_p3_s22_t20)
  MoveL (stk_p3_s22_t21)
  MoveL (stk_p3_s22_t22)
  MoveL (stk_p3_s22_t23)
  MoveL (stk_p3_s22_t24)
  MoveL (stk_p3_s22_t25)
  Set IO_21=0.0
  Set IO_22=0.0
  Set IO_23=0.0
  Set IO_24=0.0
  Set Tool: fbx_5_slot_05_fo6_roundShape_outPaintBrush
  Stroke stk_p3_s23
  Set IO_45=0.0
  Set IO_46=0.0
  Set IO_47=0.0
  Set IO_48=0.0
  MoveJ (stk_p3_s23_t0)
  Set IO_46=0.14000000059604645
  Set IO_47=0.14000000059604645
  MoveL (stk_p3_s23_t0)
  MoveL (stk_p3_s23_t1)
  MoveL (stk_p3_s23_t2)
  MoveL (stk_p3_s23_t3)
  MoveL (stk_p3_s23_t4)
  MoveL (stk_p3_s23_t5)
  MoveL (stk_p3_s23_t6)
  MoveL (stk_p3_s23_t7)
  MoveL (stk_p3_s23_t8)
  MoveL (stk_p3_s23_t9)
  MoveL (stk_p3_s23_t10)
  MoveL (stk_p3_s23_t11)
  MoveL (stk_p3_s23_t12)
  MoveL (stk_p3_s23_t13)
  MoveL (stk_p3_s23_t14)
  MoveL (stk_p3_s23_t15)
  MoveL (stk_p3_s23_t16)
  MoveL (stk_p3_s23_t17)
  MoveL (stk_p3_s23_t18)
  MoveL (stk_p3_s23_t19)
  MoveL (stk_p3_s23_t20)
  MoveL (stk_p3_s23_t21)
  MoveL (stk_p3_s23_t22)
  MoveL (stk_p3_s23_t23)
  MoveL (stk_p3_s23_t24)
  MoveL (stk_p3_s23_t25)
  Set IO_21=0.0
  Set IO_22=0.0
  Set IO_23=0.0
  Set IO_24=0.0
  Set Tool: fbx_5_slot_05_fo6_roundShape_outPaintBrush
  Stroke stk_p3_s24
  Set IO_45=0.0
  Set IO_46=0.0
  Set IO_47=0.0
  Set IO_48=0.0
  MoveJ (stk_p3_s24_t0)
  Set IO_46=0.14000000059604645
  MoveL (stk_p3_s24_t0)
  MoveL (stk_p3_s24_t1)
  MoveL (stk_p3_s24_t2)
  MoveL (stk_p3_s24_t3)
  MoveL (stk_p3_s24_t4)
  MoveL (stk_p3_s24_t5)
  MoveL (stk_p3_s24_t6)
  MoveL (stk_p3_s24_t7)
  MoveL (stk_p3_s24_t8)
  MoveL (stk_p3_s24_t9)
  MoveL (stk_p3_s24_t10)
  MoveL (stk_p3_s24_t11)
  MoveL (stk_p3_s24_t12)
  MoveL (stk_p3_s24_t13)
  MoveL (stk_p3_s24_t14)
  MoveL (stk_p3_s24_t15)
  MoveL (stk_p3_s24_t16)
  MoveL (stk_p3_s24_t17)
  MoveL (stk_p3_s24_t18)
  MoveL (stk_p3_s24_t19)
  MoveL (stk_p3_s24_t20)
  MoveL (stk_p3_s24_t21)
  MoveL (stk_p3_s24_t22)
  MoveL (stk_p3_s24_t23)
  MoveL (stk_p3_s24_t24)
  MoveL (stk_p3_s24_t25)
  Set IO_21=0.0
  Set IO_22=0.0
  Set IO_23=0.0
  Set IO_24=0.0
  Set Tool: fbx_5_slot_05_fo6_roundShape_outPaintBrush
  Stroke stk_p3_s25
  Set IO_45=0.0
  Set IO_46=0.0
  Set IO_47=0.0
  Set IO_48=0.0
  MoveJ (stk_p3_s25_t0)
  Set IO_45=0.14000000059604645
  Set IO_46=0.14000000059604645
  Set IO_47=0.14000000059604645
  MoveL (stk_p3_s25_t0)
  MoveL (stk_p3_s25_t1)
  MoveL (stk_p3_s25_t2)
  MoveL (stk_p3_s25_t3)
  MoveL (stk_p3_s25_t4)
  MoveL (stk_p3_s25_t5)
  MoveL (stk_p3_s25_t6)
  MoveL (stk_p3_s25_t7)
  MoveL (stk_p3_s25_t8)
  MoveL (stk_p3_s25_t9)
  MoveL (stk_p3_s25_t10)
  MoveL (stk_p3_s25_t11)
  MoveL (stk_p3_s25_t12)
  MoveL (stk_p3_s25_t13)
  MoveL (stk_p3_s25_t14)
  MoveL (stk_p3_s25_t15)
  MoveL (stk_p3_s25_t16)
  MoveL (stk_p3_s25_t17)
  MoveL (stk_p3_s25_t18)
  MoveL (stk_p3_s25_t19)
  MoveL (stk_p3_s25_t20)
  MoveL (stk_p3_s25_t21)
  MoveL (stk_p3_s25_t22)
  MoveL (stk_p3_s25_t23)
  MoveL (stk_p3_s25_t24)
  MoveL (stk_p3_s25_t25)
  Set IO_21=0.0
  Set IO_22=0.0
  Set IO_23=0.0
  Set IO_24=0.0
  Set Tool: fbx_5_slot_05_fo6_roundShape_outPaintBrush
  Stroke stk_p3_s26
  Set IO_45=0.0
  Set IO_46=0.0
  Set IO_47=0.0
  Set IO_48=0.0
  MoveJ (stk_p3_s26_t0)
  Set IO_45=0.14000000059604645
  Set IO_46=0.14000000059604645
  MoveL (stk_p3_s26_t0)
  MoveL (stk_p3_s26_t1)
  MoveL (stk_p3_s26_t2)
  MoveL (stk_p3_s26_t3)
  MoveL (stk_p3_s26_t4)
  MoveL (stk_p3_s26_t5)
  MoveL (stk_p3_s26_t6)
  MoveL (stk_p3_s26_t7)
  MoveL (stk_p3_s26_t8)
  MoveL (stk_p3_s26_t9)
  MoveL (stk_p3_s26_t10)
  MoveL (stk_p3_s26_t11)
  MoveL (stk_p3_s26_t12)
  MoveL (stk_p3_s26_t13)
  MoveL (stk_p3_s26_t14)
  MoveL (stk_p3_s26_t15)
  MoveL (stk_p3_s26_t16)
  MoveL (stk_p3_s26_t17)
  MoveL (stk_p3_s26_t18)
  MoveL (stk_p3_s26_t19)
  MoveL (stk_p3_s26_t20)
  MoveL (stk_p3_s26_t21)
  MoveL (stk_p3_s26_t22)
  MoveL (stk_p3_s26_t23)
  MoveL (stk_p3_s26_t24)
  MoveL (stk_p3_s26_t25)
  Set IO_21=0.0
  Set IO_22=0.0
  Set IO_23=0.0
  Set IO_24=0.0
  Set Tool: fbx_5_slot_05_fo6_roundShape_outPaintBrush
  Stroke stk_p3_s27
  Set IO_45=0.0
  Set IO_46=0.0
  Set IO_47=0.0
  Set IO_48=0.0
  MoveJ (stk_p3_s27_t0)
  Set IO_45=0.14000000059604645
  MoveL (stk_p3_s27_t0)
  MoveL (stk_p3_s27_t1)
  MoveL (stk_p3_s27_t2)
  MoveL (stk_p3_s27_t3)
  MoveL (stk_p3_s27_t4)
  MoveL (stk_p3_s27_t5)
  MoveL (stk_p3_s27_t6)
  MoveL (stk_p3_s27_t7)
  MoveL (stk_p3_s27_t8)
  MoveL (stk_p3_s27_t9)
  MoveL (stk_p3_s27_t10)
  MoveL (stk_p3_s27_t11)
  MoveL (stk_p3_s27_t12)
  MoveL (stk_p3_s27_t13)
  MoveL (stk_p3_s27_t14)
  MoveL (stk_p3_s27_t15)
  MoveL (stk_p3_s27_t16)
  MoveL (stk_p3_s27_t17)
  MoveL (stk_p3_s27_t18)
  MoveL (stk_p3_s27_t19)
  MoveL (stk_p3_s27_t20)
  MoveL (stk_p3_s27_t21)
  MoveL (stk_p3_s27_t22)
  MoveL (stk_p3_s27_t23)
  MoveL (stk_p3_s27_t24)
  MoveL (stk_p3_s27_t25)
  Set IO_21=0.0
  Set IO_22=0.0
  Set IO_23=0.0
  Set IO_24=0.0
  Set IO_49=1.0
  Pause 1.0 s
  Set IO_49=0.0
  MoveJ (home_approach)
